LIN {X 0,Y 467.101,Z 440.554,A -85,B 0,C 180,E1 -7437.809,E2 -7437.809} C_VEL
LIN {X 0,Y 466.895,Z 445.866,A -85,B 0,C 180,E1 -7439.217,E2 -7439.217} C_VEL
LIN {X 0,Y 466.777,Z 448.845,A -85,B 0,C 180,E1 -7440.207,E2 -7440.207} C_VEL
LIN {X 0,Y 466.674,Z 451.155,A -85,B 0,C 180,E1 -7441.19,E2 -7441.19} C_VEL
LIN {X 0,Y 466.545,Z 453.69,A -85,B 0,C 180,E1 -7442.72,E2 -7442.72} C_VEL
LIN {X 0,Y 466.485,Z 454.874,A -85,B 0,C 180,E1 -7444.093,E2 -7444.093} C_VEL
LIN {X 0,Y 466.485,Z 455.129,A -85,B 0,C 180,E1 -7445.049,E2 -7445.049} C_VEL
LIN {X 0,Y 466.511,Z 454.294,A -85,B 0,C 180,E1 -7446.776,E2 -7446.776} C_VEL
LIN {X 0,Y 466.551,Z 452.966,A -85,B 0,C 180,E1 -7447.877,E2 -7447.877} C_VEL
LIN {X 0,Y 466.7,Z 450.858,A -85,B 0,C 180,E1 -7449.013,E2 -7449.013} C_VEL
LIN {X 0,Y 466.824,Z 447.854,A -85,B 0,C 180,E1 -7450.2,E2 -7450.2} C_VEL
LIN {X 0,Y 466.968,Z 443.277,A -85,B 0,C 180,E1 -7451.575,E2 -7451.575} C_VEL
LIN {X 0,Y 467.167,Z 437.426,A -85,B 0,C 180,E1 -7452.941,E2 -7452.941} C_VEL
LIN {X 0,Y 467.539,Z 430.017,A -85,B 0,C 180,E1 -7454.302,E2 -7454.302} C_VEL
LIN {X 0,Y 467.973,Z 420.781,A -85,B 0,C 180,E1 -7455.653,E2 -7455.653} C_VEL
LIN {X 0,Y 468.422,Z 411.25,A -85,B 0,C 180,E1 -7456.773,E2 -7456.773} C_VEL
LIN {X 0,Y 468.937,Z 400.379,A -85,B 0,C 180,E1 -7457.795,E2 -7457.795} C_VEL
LIN {X 0,Y 469.51,Z 388.647,A -85,B 0,C 180,E1 -7458.67,E2 -7458.67} C_VEL
LIN {X 0,Y 469.897,Z 377.126,A -85,B 0,C 180,E1 -7459.334,E2 -7459.334} C_VEL
LIN {X 0,Y 470.249,Z 364.286,A -85,B 0,C 180,E1 -7459.879,E2 -7459.879} C_VEL
LIN {X 0,Y 470.485,Z 351.401,A -85,B 0,C 180,E1 -7460.247,E2 -7460.247} C_VEL
LIN {X 0,Y 471.239,Z 259.051,A -85,B 0,C 180,E1 -7461.693,E2 -7461.693} C_VEL
LIN {X 0,Y 468.413,Z 244.23,A -85,B 0,C 180,E1 -7462.049,E2 -7462.049} C_VEL
LIN {X 0,Y 468.927,Z 230.528,A -85,B 0,C 180,E1 -7464.841,E2 -7464.841} C_VEL
LIN {X 0,Y 468.176,Z 224.517,A -85,B 0,C 180,E1 -7466.127,E2 -7466.127} C_VEL
LIN {X 0,Y 467.658,Z 221.234,A -85,B 0,C 180,E1 -7466.877,E2 -7466.877} C_VEL
LIN {X 0,Y 467.749,Z 221.221,A -85,B 0,C 180,E1 -7468.278,E2 -7468.278} C_VEL
LIN {X 0,Y 467.852,Z 221.207,A -85,B 0,C 180,E1 -7470,E2 -7470} C_VEL
LIN {X 0,Y 467.818,Z 221.207,A -85,B 0,C 180,E1 -7472.583,E2 -7472.583} C_VEL
LIN {X 0,Y 467.708,Z 221.224,A -85,B 0,C 180,E1 -7476.038,E2 -7476.038} C_VEL
LIN {X 0,Y 467.67,Z 221.226,A -85,B 0,C 180,E1 -7478.643,E2 -7478.643} C_VEL
LIN {X 0,Y 467.659,Z 221.229,A -85,B 0,C 180,E1 -7482.145,E2 -7482.145} C_VEL
LIN {X 0,Y 467.64,Z 221.237,A -85,B 0,C 180,E1 -7485.695,E2 -7485.695} C_VEL
LIN {X 0,Y 467.622,Z 221.236,A -85,B 0,C 180,E1 -7489.308,E2 -7489.308} C_VEL
LIN {X 0,Y 467.536,Z 221.245,A -85,B 0,C 180,E1 -7492.073,E2 -7492.073} C_VEL
LIN {X 0,Y 467.57,Z 221.241,A -85,B 0,C 180,E1 -7494.889,E2 -7494.889} C_VEL
LIN {X 0,Y 467.581,Z 221.243,A -85,B 0,C 180,E1 -7497.771,E2 -7497.771} C_VEL
LIN {X 0,Y 467.569,Z 221.242,A -85,B 0,C 180,E1 -7501.044,E2 -7501.044} C_VEL
LIN {X 0,Y 467.588,Z 221.238,A -85,B 0,C 180,E1 -7504.242,E2 -7504.242} C_VEL
LIN {X 0,Y 467.543,Z 221.245,A -85,B 0,C 180,E1 -7507.185,E2 -7507.185} C_VEL
LIN {X 0,Y 467.572,Z 221.24,A -85,B 0,C 180,E1 -7510.265,E2 -7510.265} C_VEL
LIN {X 0,Y 467.548,Z 221.246,A -85,B 0,C 180,E1 -7513.745,E2 -7513.745} C_VEL
LIN {X 0,Y 467.55,Z 221.243,A -85,B 0,C 180,E1 -7516.255,E2 -7516.255} C_VEL
LIN {X 0,Y 467.577,Z 221.241,A -85,B 0,C 180,E1 -7518.723,E2 -7518.723} C_VEL
LIN {X 0,Y 467.564,Z 221.242,A -85,B 0,C 180,E1 -7521.955,E2 -7521.955} C_VEL
LIN {X 0,Y 467.566,Z 221.243,A -85,B 0,C 180,E1 -7525.167,E2 -7525.167} C_VEL
LIN {X 0,Y 467.581,Z 221.24,A -85,B 0,C 180,E1 -7528.26,E2 -7528.26} C_VEL
LIN {X 0,Y 467.575,Z 221.242,A -85,B 0,C 180,E1 -7531.25,E2 -7531.25} C_VEL
LIN {X 0,Y 467.608,Z 221.236,A -85,B 0,C 180,E1 -7534.16,E2 -7534.16} C_VEL
LIN {X 0,Y 467.575,Z 221.242,A -85,B 0,C 180,E1 -7536.996,E2 -7536.996} C_VEL
LIN {X 0,Y 467.62,Z 221.236,A -85,B 0,C 180,E1 -7539.777,E2 -7539.777} C_VEL
LIN {X 0,Y 467.604,Z 221.238,A -85,B 0,C 180,E1 -7542.506,E2 -7542.506} C_VEL
LIN {X 0,Y 467.604,Z 221.239,A -85,B 0,C 180,E1 -7545.196,E2 -7545.196} C_VEL
LIN {X 0,Y 467.653,Z 221.231,A -85,B 0,C 180,E1 -7547.854,E2 -7547.854} C_VEL
LIN {X 0,Y 467.679,Z 221.23,A -85,B 0,C 180,E1 -7551.357,E2 -7551.357} C_VEL
LIN {X 0,Y 467.743,Z 221.22,A -85,B 0,C 180,E1 -7553.963,E2 -7553.963} C_VEL
LIN {X 0,Y 467.857,Z 221.207,A -85,B 0,C 180,E1 -7557.417,E2 -7557.417} C_VEL
LIN {X 0,Y 467.879,Z 221.202,A -85,B 0,C 180,E1 -7560,E2 -7560} C_VEL
LIN {X 0,Y 467.857,Z 221.208,A -85,B 0,C 180,E1 -7562.583,E2 -7562.583} C_VEL
LIN {X 0,Y 467.743,Z 221.219,A -85,B 0,C 180,E1 -7566.037,E2 -7566.037} C_VEL
LIN {X 0,Y 467.678,Z 221.232,A -85,B 0,C 180,E1 -7568.643,E2 -7568.643} C_VEL
LIN {X 0,Y 467.653,Z 221.231,A -85,B 0,C 180,E1 -7572.146,E2 -7572.146} C_VEL
LIN {X 0,Y 467.636,Z 221.233,A -85,B 0,C 180,E1 -7575.695,E2 -7575.695} C_VEL
LIN {X 0,Y 467.615,Z 221.239,A -85,B 0,C 180,E1 -7578.765,E2 -7578.765} C_VEL
LIN {X 0,Y 467.578,Z 221.241,A -85,B 0,C 180,E1 -7581.269,E2 -7581.269} C_VEL
LIN {X 0,Y 467.571,Z 221.24,A -85,B 0,C 180,E1 -7583.943,E2 -7583.943} C_VEL
LIN {X 0,Y 467.614,Z 221.238,A -85,B 0,C 180,E1 -7586.8,E2 -7586.8} C_VEL
LIN {X 0,Y 467.552,Z 221.242,A -85,B 0,C 180,E1 -7589.738,E2 -7589.738} C_VEL
LIN {X 0,Y 467.581,Z 221.243,A -85,B 0,C 180,E1 -7592.759,E2 -7592.759} C_VEL
LIN {X 0,Y 467.554,Z 221.242,A -85,B 0,C 180,E1 -7595.89,E2 -7595.89} C_VEL
LIN {X 0,Y 467.58,Z 221.24,A -85,B 0,C 180,E1 -7599.145,E2 -7599.145} C_VEL
LIN {X 0,Y 467.585,Z 221.244,A -85,B 0,C 180,E1 -7602.567,E2 -7602.567} C_VEL
LIN {X 0,Y 467.569,Z 221.241,A -85,B 0,C 180,E1 -7605.053,E2 -7605.053} C_VEL
LIN {X 0,Y 467.588,Z 221.237,A -85,B 0,C 180,E1 -7607.44,E2 -7607.44} C_VEL
LIN {X 0,Y 467.581,Z 221.241,A -85,B 0,C 180,E1 -7610.856,E2 -7610.856} C_VEL
LIN {X 0,Y 467.557,Z 221.244,A -85,B 0,C 180,E1 -7614.262,E2 -7614.262} C_VEL
LIN {X 0,Y 467.582,Z 221.238,A -85,B 0,C 180,E1 -7617.321,E2 -7617.321} C_VEL
LIN {X 0,Y 467.569,Z 221.246,A -85,B 0,C 180,E1 -7620.668,E2 -7620.668} C_VEL
LIN {X 0,Y 467.587,Z 221.244,A -85,B 0,C 180,E1 -7623.198,E2 -7623.198} C_VEL
LIN {X 0,Y 467.648,Z 221.415,A -85,B 0,C 180,E1 -7624.383,E2 -7624.383} C_VEL
LIN {X 0,Y 469.778,Z 233.014,A -85,B 0,C 180,E1 -7626.644,E2 -7626.644} C_VEL
LIN {X 0,Y 469.201,Z 246.955,A -85,B 0,C 180,E1 -7629.161,E2 -7629.161} C_VEL
LIN {X 0,Y 468.484,Z 264.68,A -85,B 0,C 180,E1 -7632.315,E2 -7632.315} C_VEL
LIN {X 0,Y 468.326,Z 268.709,A -85,B 0,C 180,E1 -7633.001,E2 -7633.001} C_VEL
LIN {X 0,Y 471.206,Z 287.43,A -85,B 0,C 180,E1 -7633.4,E2 -7633.4} C_VEL
LIN {X 0,Y 470.468,Z 376.468,A -85,B 0,C 180,E1 -7634.79,E2 -7634.79} C_VEL
LIN {X 0,Y 470.15,Z 389.788,A -85,B 0,C 180,E1 -7635.168,E2 -7635.168} C_VEL
LIN {X 0,Y 469.684,Z 402.549,A -85,B 0,C 180,E1 -7635.706,E2 -7635.706} C_VEL
LIN {X 0,Y 469.237,Z 413.892,A -85,B 0,C 180,E1 -7636.356,E2 -7636.356} C_VEL
LIN {X 0,Y 468.679,Z 425.815,A -85,B 0,C 180,E1 -7637.241,E2 -7637.241} C_VEL
LIN {X 0,Y 468.248,Z 436.107,A -85,B 0,C 180,E1 -7638.2,E2 -7638.2} C_VEL
LIN {X 0,Y 467.781,Z 444.702,A -85,B 0,C 180,E1 -7639.176,E2 -7639.176} C_VEL
LIN {X 0,Y 467.436,Z 452.63,A -85,B 0,C 180,E1 -7640.262,E2 -7640.262} C_VEL
LIN {X 0,Y 467.111,Z 460.375,A -85,B 0,C 180,E1 -7641.565,E2 -7641.565} C_VEL
LIN {X 0,Y 466.852,Z 467.499,A -85,B 0,C 180,E1 -7643.083,E2 -7643.083} C_VEL
LIN {X 0,Y 466.76,Z 472.241,A -85,B 0,C 180,E1 -7644.384,E2 -7644.384} C_VEL
LIN {X 0,Y 466.646,Z 475.861,A -85,B 0,C 180,E1 -7645.682,E2 -7645.682} C_VEL
LIN {X 0,Y 466.688,Z 477.732,A -85,B 0,C 180,E1 -7646.547,E2 -7646.547} C_VEL
LIN {X 0,Y 466.662,Z 479.133,A -85,B 0,C 180,E1 -7647.411,E2 -7647.411} C_VEL
LIN {X 0,Y 466.619,Z 480.737,A -85,B 0,C 180,E1 -7649.137,E2 -7649.137} C_VEL
LIN {X 0,Y 466.6,Z 480.953,A -85,B 0,C 180,E1 -7650,E2 -7650} C_VEL
LIN {X 0,Y 466.619,Z 480.735,A -85,B 0,C 180,E1 -7650.863,E2 -7650.863} C_VEL
LIN {X 0,Y 466.662,Z 479.123,A -85,B 0,C 180,E1 -7652.59,E2 -7652.59} C_VEL
LIN {X 0,Y 466.688,Z 477.721,A -85,B 0,C 180,E1 -7653.454,E2 -7653.454} C_VEL
LIN {X 0,Y 466.688,Z 474.771,A -85,B 0,C 180,E1 -7654.751,E2 -7654.751} C_VEL
LIN {X 0,Y 466.75,Z 470.782,A -85,B 0,C 180,E1 -7656.05,E2 -7656.05} C_VEL
LIN {X 0,Y 466.942,Z 464.65,A -85,B 0,C 180,E1 -7657.568,E2 -7657.568} C_VEL
LIN {X 0,Y 467.217,Z 457.952,A -85,B 0,C 180,E1 -7658.87,E2 -7658.87} C_VEL
LIN {X 0,Y 467.546,Z 449.643,A -85,B 0,C 180,E1 -7660.173,E2 -7660.173} C_VEL
LIN {X 0,Y 468.016,Z 441.127,A -85,B 0,C 180,E1 -7661.257,E2 -7661.257} C_VEL
LIN {X 0,Y 468.511,Z 431.038,A -85,B 0,C 180,E1 -7662.302,E2 -7662.302} C_VEL
LIN {X 0,Y 468.935,Z 420.195,A -85,B 0,C 180,E1 -7663.212,E2 -7663.212} C_VEL
LIN {X 0,Y 469.459,Z 408.784,A -85,B 0,C 180,E1 -7663.969,E2 -7663.969} C_VEL
LIN {X 0,Y 469.892,Z 397.043,A -85,B 0,C 180,E1 -7664.564,E2 -7664.564} C_VEL
LIN {X 0,Y 470.35,Z 383.529,A -85,B 0,C 180,E1 -7665.047,E2 -7665.047} C_VEL
LIN {X 0,Y 470.646,Z 370.034,A -85,B 0,C 180,E1 -7665.343,E2 -7665.343} C_VEL
LIN {X 0,Y 471.145,Z 285.886,A -85,B 0,C 180,E1 -7666.649,E2 -7666.649} C_VEL
LIN {X 0,Y 468.3,Z 268.124,A -85,B 0,C 180,E1 -7667.05,E2 -7667.05} C_VEL
LIN {X 0,Y 468.908,Z 251.671,A -85,B 0,C 180,E1 -7669.936,E2 -7669.936} C_VEL
LIN {X 0,Y 469.636,Z 234.97,A -85,B 0,C 180,E1 -7672.898,E2 -7672.898} C_VEL
LIN {X 0,Y 469.472,Z 231.104,A -85,B 0,C 180,E1 -7673.606,E2 -7673.606} C_VEL
LIN {X 0,Y 467.615,Z 221.24,A -85,B 0,C 180,E1 -7675.512,E2 -7675.512} C_VEL
LIN {X 0,Y 467.617,Z 221.239,A -85,B 0,C 180,E1 -7677.769,E2 -7677.769} C_VEL
LIN {X 0,Y 467.569,Z 221.245,A -85,B 0,C 180,E1 -7681.045,E2 -7681.045} C_VEL
LIN {X 0,Y 467.589,Z 221.238,A -85,B 0,C 180,E1 -7684.242,E2 -7684.242} C_VEL
LIN {X 0,Y 467.543,Z 221.249,A -85,B 0,C 180,E1 -7687.185,E2 -7687.185} C_VEL
LIN {X 0,Y 467.575,Z 221.237,A -85,B 0,C 180,E1 -7690.265,E2 -7690.265} C_VEL
LIN {X 0,Y 467.587,Z 221.237,A -85,B 0,C 180,E1 -7692.567,E2 -7692.567} C_VEL
LIN {X 0,Y 467.571,Z 221.244,A -85,B 0,C 180,E1 -7695.053,E2 -7695.053} C_VEL
LIN {X 0,Y 467.589,Z 221.239,A -85,B 0,C 180,E1 -7697.44,E2 -7697.44} C_VEL
LIN {X 0,Y 467.576,Z 221.242,A -85,B 0,C 180,E1 -7700.855,E2 -7700.855} C_VEL
LIN {X 0,Y 467.562,Z 221.238,A -85,B 0,C 180,E1 -7704.26,E2 -7704.26} C_VEL
LIN {X 0,Y 467.581,Z 221.24,A -85,B 0,C 180,E1 -7707.321,E2 -7707.321} C_VEL
LIN {X 0,Y 467.57,Z 221.241,A -85,B 0,C 180,E1 -7710.667,E2 -7710.667} C_VEL
LIN {X 0,Y 467.616,Z 221.237,A -85,B 0,C 180,E1 -7713.2,E2 -7713.2} C_VEL
LIN {X 0,Y 467.592,Z 221.236,A -85,B 0,C 180,E1 -7716.468,E2 -7716.468} C_VEL
LIN {X 0,Y 467.622,Z 221.232,A -85,B 0,C 180,E1 -7719.777,E2 -7719.777} C_VEL
LIN {X 0,Y 467.606,Z 221.233,A -85,B 0,C 180,E1 -7722.507,E2 -7722.507} C_VEL
LIN {X 0,Y 467.606,Z 221.234,A -85,B 0,C 180,E1 -7725.196,E2 -7725.196} C_VEL
LIN {X 0,Y 467.655,Z 221.227,A -85,B 0,C 180,E1 -7727.855,E2 -7727.855} C_VEL
LIN {X 0,Y 467.681,Z 221.226,A -85,B 0,C 180,E1 -7731.357,E2 -7731.357} C_VEL
LIN {X 0,Y 467.734,Z 221.217,A -85,B 0,C 180,E1 -7733.963,E2 -7733.963} C_VEL
LIN {X 0,Y 467.859,Z 221.204,A -85,B 0,C 180,E1 -7737.417,E2 -7737.417} C_VEL
LIN {X 0,Y 467.881,Z 221.196,A -85,B 0,C 180,E1 -7740,E2 -7740} C_VEL
LIN {X 0,Y 467.858,Z 221.208,A -85,B 0,C 180,E1 -7742.583,E2 -7742.583} C_VEL
LIN {X 0,Y 467.734,Z 221.219,A -85,B 0,C 180,E1 -7746.038,E2 -7746.038} C_VEL
LIN {X 0,Y 467.681,Z 221.228,A -85,B 0,C 180,E1 -7748.643,E2 -7748.643} C_VEL
LIN {X 0,Y 467.655,Z 221.226,A -85,B 0,C 180,E1 -7752.146,E2 -7752.146} C_VEL
LIN {X 0,Y 467.639,Z 221.228,A -85,B 0,C 180,E1 -7755.695,E2 -7755.695} C_VEL
LIN {X 0,Y 467.617,Z 221.238,A -85,B 0,C 180,E1 -7758.765,E2 -7758.765} C_VEL
LIN {X 0,Y 467.58,Z 221.238,A -85,B 0,C 180,E1 -7761.268,E2 -7761.268} C_VEL
LIN {X 0,Y 467.563,Z 221.24,A -85,B 0,C 180,E1 -7763.944,E2 -7763.944} C_VEL
LIN {X 0,Y 467.565,Z 221.245,A -85,B 0,C 180,E1 -7766.804,E2 -7766.804} C_VEL
LIN {X 0,Y 467.547,Z 221.24,A -85,B 0,C 180,E1 -7769.739,E2 -7769.739} C_VEL
LIN {X 0,Y 467.579,Z 221.243,A -85,B 0,C 180,E1 -7772.759,E2 -7772.759} C_VEL
LIN {X 0,Y 467.549,Z 221.246,A -85,B 0,C 180,E1 -7775.89,E2 -7775.89} C_VEL
LIN {X 0,Y 467.547,Z 221.245,A -85,B 0,C 180,E1 -7779.149,E2 -7779.149} C_VEL
LIN {X 0,Y 467.564,Z 221.243,A -85,B 0,C 180,E1 -7781.405,E2 -7781.405} C_VEL
LIN {X 0,Y 467.564,Z 221.31,A -85,B 0,C 180,E1 -7783.521,E2 -7783.521} C_VEL
LIN {X 0,Y 468.843,Z 228.525,A -85,B 0,C 180,E1 -7785.001,E2 -7785.001} C_VEL
LIN {X 0,Y 468.462,Z 244.324,A -85,B 0,C 180,E1 -7788.025,E2 -7788.025} C_VEL
LIN {X 0,Y 471.369,Z 259.441,A -85,B 0,C 180,E1 -7788.378,E2 -7788.378} C_VEL
LIN {X 0,Y 470.565,Z 351.674,A -85,B 0,C 180,E1 -7789.824,E2 -7789.824} C_VEL
LIN {X 0,Y 470.284,Z 365.391,A -85,B 0,C 180,E1 -7790.223,E2 -7790.223} C_VEL
LIN {X 0,Y 469.973,Z 377.504,A -85,B 0,C 180,E1 -7790.747,E2 -7790.747} C_VEL
LIN {X 0,Y 469.481,Z 389.628,A -85,B 0,C 180,E1 -7791.456,E2 -7791.456} C_VEL
LIN {X 0,Y 469.023,Z 400.201,A -85,B 0,C 180,E1 -7792.251,E2 -7792.251} C_VEL
LIN {X 0,Y 468.509,Z 411.002,A -85,B 0,C 180,E1 -7793.262,E2 -7793.262} C_VEL
LIN {X 0,Y 468.031,Z 420.88,A -85,B 0,C 180,E1 -7794.42,E2 -7794.42} C_VEL
LIN {X 0,Y 467.78,Z 426.185,A -85,B 0,C 180,E1 -7795.161,E2 -7795.161} C_VEL
LIN {X 0,Y 467.008,Z 429.892,A -85,B 0,C 180,E1 -7795.717,E2 -7795.717} C_VEL
LIN {X 0,Y 463.897,Z 435.547,A -85,B 0,C 180,E1 -7796.645,E2 -7796.645} C_VEL
LIN {X 0,Y 460.752,Z 440.515,A -85,B 0,C 180,E1 -7797.639,E2 -7797.639} C_VEL
LIN {X 0,Y 459.944,Z 443.146,A -85,B 0,C 180,E1 -7798.292,E2 -7798.292} C_VEL
LIN {X 0,Y 459.792,Z 447.857,A -85,B 0,C 180,E1 -7799.708,E2 -7799.708} C_VEL
LIN {X 0,Y 459.658,Z 450.452,A -85,B 0,C 180,E1 -7800.708,E2 -7800.708} C_VEL
LIN {X 0,Y 459.525,Z 452.445,A -85,B 0,C 180,E1 -7801.698,E2 -7801.698} C_VEL
LIN {X 0,Y 459.464,Z 453.893,A -85,B 0,C 180,E1 -7802.685,E2 -7802.685} C_VEL
LIN {X 0,Y 459.408,Z 454.848,A -85,B 0,C 180,E1 -7803.664,E2 -7803.664} C_VEL
LIN {X 0,Y 459.416,Z 455.261,A -85,B 0,C 180,E1 -7804.638,E2 -7804.638} C_VEL
LIN {X 0,Y 459.386,Z 455.226,A -85,B 0,C 180,E1 -7805.603,E2 -7805.603} C_VEL
LIN {X 0,Y 459.418,Z 454.657,A -85,B 0,C 180,E1 -7806.615,E2 -7806.615} C_VEL
LIN {X 0,Y 459.429,Z 453.7,A -85,B 0,C 180,E1 -7807.516,E2 -7807.516} C_VEL
LIN {X 0,Y 459.585,Z 451.44,A -85,B 0,C 180,E1 -7808.879,E2 -7808.879} C_VEL
LIN {X 0,Y 459.752,Z 447.841,A -85,B 0,C 180,E1 -7810.348,E2 -7810.348} C_VEL
LIN {X 0,Y 459.909,Z 443.083,A -85,B 0,C 180,E1 -7811.777,E2 -7811.777} C_VEL
LIN {X 0,Y 460.145,Z 437.274,A -85,B 0,C 180,E1 -7813.13,E2 -7813.13} C_VEL
LIN {X 0,Y 460.539,Z 429.763,A -85,B 0,C 180,E1 -7814.511,E2 -7814.511} C_VEL
LIN {X 0,Y 461.007,Z 420.437,A -85,B 0,C 180,E1 -7815.882,E2 -7815.882} C_VEL
LIN {X 0,Y 461.567,Z 410.599,A -85,B 0,C 180,E1 -7817.032,E2 -7817.032} C_VEL
LIN {X 0,Y 462.057,Z 399.903,A -85,B 0,C 180,E1 -7818.039,E2 -7818.039} C_VEL
LIN {X 0,Y 462.564,Z 389.426,A -85,B 0,C 180,E1 -7818.83,E2 -7818.83} C_VEL
LIN {X 0,Y 463.044,Z 376.849,A -85,B 0,C 180,E1 -7819.567,E2 -7819.567} C_VEL
LIN {X 0,Y 463.389,Z 363.758,A -85,B 0,C 180,E1 -7820.124,E2 -7820.124} C_VEL
LIN {X 0,Y 463.647,Z 351.397,A -85,B 0,C 180,E1 -7820.475,E2 -7820.475} C_VEL
LIN {X 0,Y 464.461,Z 260.073,A -85,B 0,C 180,E1 -7821.924,E2 -7821.924} C_VEL
LIN {X 0,Y 461.465,Z 244.435,A -85,B 0,C 180,E1 -7822.302,E2 -7822.302} C_VEL
LIN {X 0,Y 461.918,Z 230.419,A -85,B 0,C 180,E1 -7825.2,E2 -7825.2} C_VEL
LIN {X 0,Y 460.644,Z 222.108,A -85,B 0,C 180,E1 -7827.048,E2 -7827.048} C_VEL
LIN {X 0,Y 460.822,Z 222.083,A -85,B 0,C 180,E1 -7830,E2 -7830} C_VEL
LIN {X 0,Y 460.762,Z 222.086,A -85,B 0,C 180,E1 -7832.623,E2 -7832.623} C_VEL
LIN {X 0,Y 460.674,Z 222.1,A -85,B 0,C 180,E1 -7836.13,E2 -7836.13} C_VEL
LIN {X 0,Y 460.62,Z 222.105,A -85,B 0,C 180,E1 -7838.776,E2 -7838.776} C_VEL
LIN {X 0,Y 460.6,Z 222.108,A -85,B 0,C 180,E1 -7842.435,E2 -7842.435} C_VEL
LIN {X 0,Y 460.581,Z 222.113,A -85,B 0,C 180,E1 -7845.988,E2 -7845.988} C_VEL
LIN {X 0,Y 460.569,Z 222.118,A -85,B 0,C 180,E1 -7849.615,E2 -7849.615} C_VEL
LIN {X 0,Y 460.512,Z 222.119,A -85,B 0,C 180,E1 -7852.428,E2 -7852.428} C_VEL
LIN {X 0,Y 460.549,Z 222.119,A -85,B 0,C 180,E1 -7855.796,E2 -7855.796} C_VEL
LIN {X 0,Y 460.528,Z 222.118,A -85,B 0,C 180,E1 -7858.234,E2 -7858.234} C_VEL
LIN {X 0,Y 460.521,Z 222.12,A -85,B 0,C 180,E1 -7861.282,E2 -7861.282} C_VEL
LIN {X 0,Y 460.531,Z 222.117,A -85,B 0,C 180,E1 -7864.505,E2 -7864.505} C_VEL
LIN {X 0,Y 460.499,Z 222.126,A -85,B 0,C 180,E1 -7867.623,E2 -7867.623} C_VEL
LIN {X 0,Y 460.536,Z 222.117,A -85,B 0,C 180,E1 -7870.268,E2 -7870.268} C_VEL
LIN {X 0,Y 460.508,Z 222.123,A -85,B 0,C 180,E1 -7873.374,E2 -7873.374} C_VEL
LIN {X 0,Y 460.496,Z 222.123,A -85,B 0,C 180,E1 -7876.624,E2 -7876.624} C_VEL
LIN {X 0,Y 460.538,Z 222.12,A -85,B 0,C 180,E1 -7879.731,E2 -7879.731} C_VEL
LIN {X 0,Y 460.499,Z 222.122,A -85,B 0,C 180,E1 -7882.523,E2 -7882.523} C_VEL
LIN {X 0,Y 460.547,Z 222.119,A -85,B 0,C 180,E1 -7885.624,E2 -7885.624} C_VEL
LIN {X 0,Y 460.535,Z 222.119,A -85,B 0,C 180,E1 -7888.744,E2 -7888.744} C_VEL
LIN {X 0,Y 460.579,Z 222.112,A -85,B 0,C 180,E1 -7892.253,E2 -7892.253} C_VEL
LIN {X 0,Y 460.557,Z 222.117,A -85,B 0,C 180,E1 -7894.705,E2 -7894.705} C_VEL
LIN {X 0,Y 460.509,Z 222.124,A -85,B 0,C 180,E1 -7897.571,E2 -7897.571} C_VEL
LIN {X 0,Y 460.566,Z 222.114,A -85,B 0,C 180,E1 -7900.384,E2 -7900.384} C_VEL
LIN {X 0,Y 460.562,Z 222.115,A -85,B 0,C 180,E1 -7903.146,E2 -7903.146} C_VEL
LIN {X 0,Y 460.552,Z 222.116,A -85,B 0,C 180,E1 -7905.868,E2 -7905.868} C_VEL
LIN {X 0,Y 460.609,Z 222.11,A -85,B 0,C 180,E1 -7908.559,E2 -7908.559} C_VEL
LIN {X 0,Y 460.692,Z 222.098,A -85,B 0,C 180,E1 -7912.108,E2 -7912.108} C_VEL
LIN {X 0,Y 460.696,Z 222.1,A -85,B 0,C 180,E1 -7914.748,E2 -7914.748} C_VEL
LIN {X 0,Y 460.822,Z 222.083,A -85,B 0,C 180,E1 -7917.378,E2 -7917.378} C_VEL
LIN {X 0,Y 460.85,Z 222.078,A -85,B 0,C 180,E1 -7920,E2 -7920} C_VEL
LIN {X 0,Y 460.822,Z 222.085,A -85,B 0,C 180,E1 -7922.622,E2 -7922.622} C_VEL
LIN {X 0,Y 460.709,Z 222.096,A -85,B 0,C 180,E1 -7926.13,E2 -7926.13} C_VEL
LIN {X 0,Y 460.625,Z 222.109,A -85,B 0,C 180,E1 -7928.776,E2 -7928.776} C_VEL
LIN {X 0,Y 460.61,Z 222.11,A -85,B 0,C 180,E1 -7932.445,E2 -7932.445} C_VEL
LIN {X 0,Y 460.597,Z 222.109,A -85,B 0,C 180,E1 -7935.998,E2 -7935.998} C_VEL
LIN {X 0,Y 460.568,Z 222.115,A -85,B 0,C 180,E1 -7938.902,E2 -7938.902} C_VEL
LIN {X 0,Y 460.513,Z 222.121,A -85,B 0,C 180,E1 -7941.486,E2 -7941.486} C_VEL
LIN {X 0,Y 460.54,Z 222.118,A -85,B 0,C 180,E1 -7944.332,E2 -7944.332} C_VEL
LIN {X 0,Y 460.57,Z 222.113,A -85,B 0,C 180,E1 -7947.244,E2 -7947.244} C_VEL
LIN {X 0,Y 460.508,Z 222.122,A -85,B 0,C 180,E1 -7950.24,E2 -7950.24} C_VEL
LIN {X 0,Y 460.527,Z 222.118,A -85,B 0,C 180,E1 -7953.325,E2 -7953.325} C_VEL
LIN {X 0,Y 460.476,Z 222.129,A -85,B 0,C 180,E1 -7956.53,E2 -7956.53} C_VEL
LIN {X 0,Y 460.53,Z 222.117,A -85,B 0,C 180,E1 -7959.863,E2 -7959.863} C_VEL
LIN {X 0,Y 460.512,Z 222.121,A -85,B 0,C 180,E1 -7962.901,E2 -7962.901} C_VEL
LIN {X 0,Y 460.51,Z 222.119,A -85,B 0,C 180,E1 -7965.831,E2 -7965.831} C_VEL
LIN {X 0,Y 460.53,Z 222.118,A -85,B 0,C 180,E1 -7968.989,E2 -7968.989} C_VEL
LIN {X 0,Y 460.524,Z 222.117,A -85,B 0,C 180,E1 -7971.267,E2 -7971.267} C_VEL
LIN {X 0,Y 460.508,Z 222.126,A -85,B 0,C 180,E1 -7974.555,E2 -7974.555} C_VEL
LIN {X 0,Y 460.531,Z 222.115,A -85,B 0,C 180,E1 -7977.716,E2 -7977.716} C_VEL
LIN {X 0,Y 460.539,Z 222.121,A -85,B 0,C 180,E1 -7980.769,E2 -7980.769} C_VEL
LIN {X 0,Y 460.546,Z 222.121,A -85,B 0,C 180,E1 -7983.734,E2 -7983.734} C_VEL
LIN {X 0,Y 460.575,Z 222.201,A -85,B 0,C 180,E1 -7984.153,E2 -7984.153} C_VEL
LIN {X 0,Y 462.801,Z 234.066,A -85,B 0,C 180,E1 -7986.508,E2 -7986.508} C_VEL
LIN {X 0,Y 462.24,Z 248.01,A -85,B 0,C 180,E1 -7989.066,E2 -7989.066} C_VEL
LIN {X 0,Y 461.464,Z 265.729,A -85,B 0,C 180,E1 -7992.266,E2 -7992.266} C_VEL
LIN {X 0,Y 461.339,Z 268.541,A -85,B 0,C 180,E1 -7992.741,E2 -7992.741} C_VEL
LIN {X 0,Y 464.399,Z 287.867,A -85,B 0,C 180,E1 -7993.165,E2 -7993.165} C_VEL
LIN {X 0,Y 463.577,Z 377.159,A -85,B 0,C 180,E1 -7994.587,E2 -7994.587} C_VEL
LIN {X 0,Y 463.193,Z 390.942,A -85,B 0,C 180,E1 -7994.996,E2 -7994.996} C_VEL
LIN {X 0,Y 462.761,Z 403.327,A -85,B 0,C 180,E1 -7995.544,E2 -7995.544} C_VEL
LIN {X 0,Y 462.244,Z 415.198,A -85,B 0,C 180,E1 -7996.257,E2 -7996.257} C_VEL
LIN {X 0,Y 461.692,Z 426.438,A -85,B 0,C 180,E1 -7997.122,E2 -7997.122} C_VEL
LIN {X 0,Y 461.218,Z 436.918,A -85,B 0,C 180,E1 -7998.129,E2 -7998.129} C_VEL
LIN {X 0,Y 460.682,Z 446.162,A -85,B 0,C 180,E1 -7999.229,E2 -7999.229} C_VEL
LIN {X 0,Y 460.265,Z 455.154,A -85,B 0,C 180,E1 -8000.553,E2 -8000.553} C_VEL
LIN {X 0,Y 459.951,Z 462.395,A -85,B 0,C 180,E1 -8001.875,E2 -8001.875} C_VEL
LIN {X 0,Y 459.743,Z 468.46,A -85,B 0,C 180,E1 -8003.273,E2 -8003.273} C_VEL
LIN {X 0,Y 459.649,Z 473.351,A -85,B 0,C 180,E1 -8004.736,E2 -8004.736} C_VEL
LIN {X 0,Y 459.563,Z 475.655,A -85,B 0,C 180,E1 -8005.615,E2 -8005.615} C_VEL
LIN {X 0,Y 459.583,Z 477.528,A -85,B 0,C 180,E1 -8006.493,E2 -8006.493} C_VEL
LIN {X 0,Y 459.584,Z 478.932,A -85,B 0,C 180,E1 -8007.371,E2 -8007.371} C_VEL
LIN {X 0,Y 459.522,Z 480.539,A -85,B 0,C 180,E1 -8009.124,E2 -8009.124} C_VEL
LIN {X 0,Y 459.531,Z 480.757,A -85,B 0,C 180,E1 -8010,E2 -8010} C_VEL
LIN {X 0,Y 459.522,Z 480.54,A -85,B 0,C 180,E1 -8010.876,E2 -8010.876} C_VEL
LIN {X 0,Y 459.584,Z 478.93,A -85,B 0,C 180,E1 -8012.63,E2 -8012.63} C_VEL
LIN {X 0,Y 459.583,Z 477.528,A -85,B 0,C 180,E1 -8013.507,E2 -8013.507} C_VEL
LIN {X 0,Y 459.616,Z 474.581,A -85,B 0,C 180,E1 -8014.824,E2 -8014.824} C_VEL
LIN {X 0,Y 459.714,Z 469.56,A -85,B 0,C 180,E1 -8016.431,E2 -8016.431} C_VEL
LIN {X 0,Y 459.901,Z 463.447,A -85,B 0,C 180,E1 -8017.905,E2 -8017.905} C_VEL
LIN {X 0,Y 460.212,Z 456.525,A -85,B 0,C 180,E1 -8019.227,E2 -8019.227} C_VEL
LIN {X 0,Y 460.503,Z 449.458,A -85,B 0,C 180,E1 -8020.33,E2 -8020.33} C_VEL
LIN {X 0,Y 461.029,Z 440.946,A -85,B 0,C 180,E1 -8021.43,E2 -8021.43} C_VEL
LIN {X 0,Y 461.557,Z 431.024,A -85,B 0,C 180,E1 -8022.475,E2 -8022.475} C_VEL
LIN {X 0,Y 462.011,Z 420.022,A -85,B 0,C 180,E1 -8023.414,E2 -8023.414} C_VEL
LIN {X 0,Y 462.55,Z 408.618,A -85,B 0,C 180,E1 -8024.182,E2 -8024.182} C_VEL
LIN {X 0,Y 463.021,Z 396.894,A -85,B 0,C 180,E1 -8024.785,E2 -8024.785} C_VEL
LIN {X 0,Y 463.504,Z 383.404,A -85,B 0,C 180,E1 -8025.275,E2 -8025.275} C_VEL
LIN {X 0,Y 463.818,Z 369.991,A -85,B 0,C 180,E1 -8025.574,E2 -8025.574} C_VEL
LIN {X 0,Y 464.358,Z 286.812,A -85,B 0,C 180,E1 -8026.886,E2 -8026.886} C_VEL
LIN {X 0,Y 461.349,Z 267.883,A -85,B 0,C 180,E1 -8027.327,E2 -8027.327} C_VEL
LIN {X 0,Y 462.003,Z 251.476,A -85,B 0,C 180,E1 -8030.247,E2 -8030.247} C_VEL
LIN {X 0,Y 462.779,Z 234.798,A -85,B 0,C 180,E1 -8033.257,E2 -8033.257} C_VEL
LIN {X 0,Y 461.519,Z 227.044,A -85,B 0,C 180,E1 -8034.757,E2 -8034.757} C_VEL
LIN {X 0,Y 460.559,Z 222.118,A -85,B 0,C 180,E1 -8035.743,E2 -8035.743} C_VEL
LIN {X 0,Y 460.55,Z 222.117,A -85,B 0,C 180,E1 -8038.233,E2 -8038.233} C_VEL
LIN {X 0,Y 460.522,Z 222.125,A -85,B 0,C 180,E1 -8041.283,E2 -8041.283} C_VEL
LIN {X 0,Y 460.532,Z 222.118,A -85,B 0,C 180,E1 -8044.505,E2 -8044.505} C_VEL
LIN {X 0,Y 460.499,Z 222.123,A -85,B 0,C 180,E1 -8047.623,E2 -8047.623} C_VEL
LIN {X 0,Y 460.539,Z 222.114,A -85,B 0,C 180,E1 -8050.269,E2 -8050.269} C_VEL
LIN {X 0,Y 460.509,Z 222.126,A -85,B 0,C 180,E1 -8053.374,E2 -8053.374} C_VEL
LIN {X 0,Y 460.5,Z 222.122,A -85,B 0,C 180,E1 -8056.625,E2 -8056.625} C_VEL
LIN {X 0,Y 460.539,Z 222.117,A -85,B 0,C 180,E1 -8059.731,E2 -8059.731} C_VEL
LIN {X 0,Y 460.5,Z 222.119,A -85,B 0,C 180,E1 -8062.523,E2 -8062.523} C_VEL
LIN {X 0,Y 460.548,Z 222.115,A -85,B 0,C 180,E1 -8065.624,E2 -8065.624} C_VEL
LIN {X 0,Y 460.537,Z 222.115,A -85,B 0,C 180,E1 -8068.744,E2 -8068.744} C_VEL
LIN {X 0,Y 460.581,Z 222.107,A -85,B 0,C 180,E1 -8072.254,E2 -8072.254} C_VEL
LIN {X 0,Y 460.558,Z 222.115,A -85,B 0,C 180,E1 -8074.705,E2 -8074.705} C_VEL
LIN {X 0,Y 460.51,Z 222.119,A -85,B 0,C 180,E1 -8077.571,E2 -8077.571} C_VEL
LIN {X 0,Y 460.568,Z 222.111,A -85,B 0,C 180,E1 -8080.384,E2 -8080.384} C_VEL
LIN {X 0,Y 460.563,Z 222.117,A -85,B 0,C 180,E1 -8083.146,E2 -8083.146} C_VEL
LIN {X 0,Y 460.555,Z 222.107,A -85,B 0,C 180,E1 -8085.868,E2 -8085.868} C_VEL
LIN {X 0,Y 460.61,Z 222.108,A -85,B 0,C 180,E1 -8088.559,E2 -8088.559} C_VEL
LIN {X 0,Y 460.694,Z 222.094,A -85,B 0,C 180,E1 -8092.109,E2 -8092.109} C_VEL
LIN {X 0,Y 460.693,Z 222.098,A -85,B 0,C 180,E1 -8094.748,E2 -8094.748} C_VEL
LIN {X 0,Y 460.824,Z 222.081,A -85,B 0,C 180,E1 -8097.378,E2 -8097.378} C_VEL
LIN {X 0,Y 460.852,Z 222.071,A -85,B 0,C 180,E1 -8100,E2 -8100} C_VEL
LIN {X 0,Y 460.823,Z 222.085,A -85,B 0,C 180,E1 -8102.622,E2 -8102.622} C_VEL
LIN {X 0,Y 460.7,Z 222.095,A -85,B 0,C 180,E1 -8106.13,E2 -8106.13} C_VEL
LIN {X 0,Y 460.628,Z 222.107,A -85,B 0,C 180,E1 -8108.776,E2 -8108.776} C_VEL
LIN {X 0,Y 460.613,Z 222.106,A -85,B 0,C 180,E1 -8112.445,E2 -8112.445} C_VEL
LIN {X 0,Y 460.6,Z 222.106,A -85,B 0,C 180,E1 -8115.998,E2 -8115.998} C_VEL
LIN {X 0,Y 460.57,Z 222.116,A -85,B 0,C 180,E1 -8118.902,E2 -8118.902} C_VEL
LIN {X 0,Y 460.515,Z 222.117,A -85,B 0,C 180,E1 -8121.486,E2 -8121.486} C_VEL
LIN {X 0,Y 460.53,Z 222.119,A -85,B 0,C 180,E1 -8124.333,E2 -8124.333} C_VEL
LIN {X 0,Y 460.534,Z 222.117,A -85,B 0,C 180,E1 -8127.246,E2 -8127.246} C_VEL
LIN {X 0,Y 460.507,Z 222.121,A -85,B 0,C 180,E1 -8130.24,E2 -8130.24} C_VEL
LIN {X 0,Y 460.519,Z 222.12,A -85,B 0,C 180,E1 -8133.326,E2 -8133.326} C_VEL
LIN {X 0,Y 460.465,Z 222.132,A -85,B 0,C 180,E1 -8136.531,E2 -8136.531} C_VEL
LIN {X 0,Y 460.511,Z 222.122,A -85,B 0,C 180,E1 -8139.865,E2 -8139.865} C_VEL
LIN {X 0,Y 460.52,Z 222.123,A -85,B 0,C 180,E1 -8143.222,E2 -8143.222} C_VEL
LIN {X 0,Y 460.564,Z 222.384,A -85,B 0,C 180,E1 -8143.368,E2 -8143.368} C_VEL
LIN {X 0,Y 461.929,Z 230.208,A -85,B 0,C 180,E1 -8144.985,E2 -8144.985} C_VEL
LIN {X 0,Y 461.504,Z 244.26,A -85,B 0,C 180,E1 -8147.729,E2 -8147.729} C_VEL
LIN {X 0,Y 464.597,Z 260.384,A -85,B 0,C 180,E1 -8148.134,E2 -8148.134} C_VEL
LIN {X 0,Y 463.748,Z 351.503,A -85,B 0,C 180,E1 -8149.584,E2 -8149.584} C_VEL
LIN {X 0,Y 463.438,Z 365.072,A -85,B 0,C 180,E1 -8149.978,E2 -8149.978} C_VEL
LIN {X 0,Y 463.079,Z 377.362,A -85,B 0,C 180,E1 -8150.51,E2 -8150.51} C_VEL
LIN {X 0,Y 462.605,Z 389.448,A -85,B 0,C 180,E1 -8151.221,E2 -8151.221} C_VEL
LIN {X 0,Y 462.054,Z 401.471,A -85,B 0,C 180,E1 -8152.145,E2 -8152.145} C_VEL
LIN {X 0,Y 461.524,Z 411.961,A -85,B 0,C 180,E1 -8153.159,E2 -8153.159} C_VEL
LIN {X 0,Y 460.996,Z 421.793,A -85,B 0,C 180,E1 -8154.351,E2 -8154.351} C_VEL
LIN {X 0,Y 460.55,Z 430.286,A -85,B 0,C 180,E1 -8155.624,E2 -8155.624} C_VEL
LIN {X 0,Y 460.181,Z 437.34,A -85,B 0,C 180,E1 -8156.933,E2 -8156.933} C_VEL
LIN {X 0,Y 459.944,Z 443.146,A -85,B 0,C 180,E1 -8158.292,E2 -8158.292} C_VEL
LIN {X 0,Y 459.163,Z 445.588,A -85,B 0,C 180,E1 -8158.96,E2 -8158.96} C_VEL
LIN {X 0,Y 456.126,Z 449.071,A -85,B 0,C 180,E1 -8160.062,E2 -8160.062} C_VEL
LIN {X 0,Y 453.6,Z 451.32,A -85,B 0,C 180,E1 -8160.971,E2 -8160.971} C_VEL
LIN {X 0,Y 452.502,Z 452.711,A -85,B 0,C 180,E1 -8161.686,E2 -8161.686} C_VEL
LIN {X 0,Y 452.404,Z 453.068,A -85,B 0,C 180,E1 -8161.929,E2 -8161.929} C_VEL
LIN {X 0,Y 452.322,Z 454.689,A -85,B 0,C 180,E1 -8163.219,E2 -8163.219} C_VEL
LIN {X 0,Y 452.316,Z 455.399,A -85,B 0,C 180,E1 -8164.316,E2 -8164.316} C_VEL
LIN {X 0,Y 452.288,Z 455.499,A -85,B 0,C 180,E1 -8165.194,E2 -8165.194} C_VEL
LIN {X 0,Y 452.319,Z 455.009,A -85,B 0,C 180,E1 -8166.453,E2 -8166.453} C_VEL
LIN {X 0,Y 452.406,Z 453.106,A -85,B 0,C 180,E1 -8168.11,E2 -8168.11} C_VEL
LIN {X 0,Y 452.592,Z 450.299,A -85,B 0,C 180,E1 -8169.55,E2 -8169.55} C_VEL
LIN {X 0,Y 452.789,Z 445.564,A -85,B 0,C 180,E1 -8171.231,E2 -8171.231} C_VEL
LIN {X 0,Y 452.981,Z 440.297,A -85,B 0,C 180,E1 -8172.623,E2 -8172.623} C_VEL
LIN {X 0,Y 453.353,Z 433.072,A -85,B 0,C 180,E1 -8174.107,E2 -8174.107} C_VEL
LIN {X 0,Y 453.78,Z 425.055,A -85,B 0,C 180,E1 -8175.423,E2 -8175.423} C_VEL
LIN {X 0,Y 454.261,Z 416.388,A -85,B 0,C 180,E1 -8176.581,E2 -8176.581} C_VEL
LIN {X 0,Y 454.778,Z 406.837,A -85,B 0,C 180,E1 -8177.618,E2 -8177.618} C_VEL
LIN {X 0,Y 455.292,Z 396.415,A -85,B 0,C 180,E1 -8178.537,E2 -8178.537} C_VEL
LIN {X 0,Y 455.935,Z 383.933,A -85,B 0,C 180,E1 -8179.402,E2 -8179.402} C_VEL
LIN {X 0,Y 456.335,Z 371.565,A -85,B 0,C 180,E1 -8180.045,E2 -8180.045} C_VEL
LIN {X 0,Y 456.68,Z 359.131,A -85,B 0,C 180,E1 -8180.505,E2 -8180.505} C_VEL
LIN {X 0,Y 456.941,Z 346.257,A -85,B 0,C 180,E1 -8180.805,E2 -8180.805} C_VEL
LIN {X 0,Y 457.619,Z 260.885,A -85,B 0,C 180,E1 -8182.168,E2 -8182.168} C_VEL
LIN {X 0,Y 454.526,Z 244.536,A -85,B 0,C 180,E1 -8182.583,E2 -8182.583} C_VEL
LIN {X 0,Y 454.999,Z 232.377,A -85,B 0,C 180,E1 -8185.127,E2 -8185.127} C_VEL
LIN {X 0,Y 453.692,Z 222.974,A -85,B 0,C 180,E1 -8187.225,E2 -8187.225} C_VEL
LIN {X 0,Y 453.792,Z 222.958,A -85,B 0,C 180,E1 -8190,E2 -8190} C_VEL
LIN {X 0,Y 453.709,Z 222.965,A -85,B 0,C 180,E1 -8192.663,E2 -8192.663} C_VEL
LIN {X 0,Y 453.641,Z 222.975,A -85,B 0,C 180,E1 -8196.226,E2 -8196.226} C_VEL
LIN {X 0,Y 453.586,Z 222.981,A -85,B 0,C 180,E1 -8198.913,E2 -8198.913} C_VEL
LIN {X 0,Y 453.567,Z 222.984,A -85,B 0,C 180,E1 -8202.529,E2 -8202.529} C_VEL
LIN {X 0,Y 453.54,Z 222.988,A -85,B 0,C 180,E1 -8206.196,E2 -8206.196} C_VEL
LIN {X 0,Y 453.519,Z 222.991,A -85,B 0,C 180,E1 -8209.039,E2 -8209.039} C_VEL
LIN {X 0,Y 453.478,Z 222.999,A -85,B 0,C 180,E1 -8211.836,E2 -8211.836} C_VEL
LIN {X 0,Y 453.495,Z 222.994,A -85,B 0,C 180,E1 -8214.735,E2 -8214.735} C_VEL
LIN {X 0,Y 453.508,Z 222.994,A -85,B 0,C 180,E1 -8217.953,E2 -8217.953} C_VEL
LIN {X 0,Y 453.476,Z 222.997,A -85,B 0,C 180,E1 -8220.759,E2 -8220.759} C_VEL
LIN {X 0,Y 453.477,Z 222.998,A -85,B 0,C 180,E1 -8223.912,E2 -8223.912} C_VEL
LIN {X 0,Y 453.45,Z 223.001,A -85,B 0,C 180,E1 -8227.189,E2 -8227.189} C_VEL
LIN {X 0,Y 453.493,Z 222.995,A -85,B 0,C 180,E1 -8230.609,E2 -8230.609} C_VEL
LIN {X 0,Y 453.46,Z 222.999,A -85,B 0,C 180,E1 -8234.221,E2 -8234.221} C_VEL
LIN {X 0,Y 453.46,Z 222.999,A -85,B 0,C 180,E1 -8237.004,E2 -8237.004} C_VEL
LIN {X 0,Y 453.493,Z 222.997,A -85,B 0,C 180,E1 -8239.409,E2 -8239.409} C_VEL
LIN {X 0,Y 453.449,Z 223,A -85,B 0,C 180,E1 -8242.227,E2 -8242.227} C_VEL
LIN {X 0,Y 453.487,Z 222.997,A -85,B 0,C 180,E1 -8245.222,E2 -8245.222} C_VEL
LIN {X 0,Y 453.464,Z 222.999,A -85,B 0,C 180,E1 -8248.474,E2 -8248.474} C_VEL
LIN {X 0,Y 453.53,Z 222.991,A -85,B 0,C 180,E1 -8252.04,E2 -8252.04} C_VEL
LIN {X 0,Y 453.512,Z 222.994,A -85,B 0,C 180,E1 -8255.265,E2 -8255.265} C_VEL
LIN {X 0,Y 453.478,Z 222.997,A -85,B 0,C 180,E1 -8258.415,E2 -8258.415} C_VEL
LIN {X 0,Y 453.519,Z 222.992,A -85,B 0,C 180,E1 -8261.008,E2 -8261.008} C_VEL
LIN {X 0,Y 453.566,Z 222.986,A -85,B 0,C 180,E1 -8263.879,E2 -8263.879} C_VEL
LIN {X 0,Y 453.561,Z 222.988,A -85,B 0,C 180,E1 -8267.471,E2 -8267.471} C_VEL
LIN {X 0,Y 453.59,Z 222.984,A -85,B 0,C 180,E1 -8271.086,E2 -8271.086} C_VEL
LIN {X 0,Y 453.676,Z 222.973,A -85,B 0,C 180,E1 -8273.775,E2 -8273.775} C_VEL
LIN {X 0,Y 453.762,Z 222.962,A -85,B 0,C 180,E1 -8277.337,E2 -8277.337} C_VEL
LIN {X 0,Y 453.82,Z 222.954,A -85,B 0,C 180,E1 -8280,E2 -8280} C_VEL
LIN {X 0,Y 453.762,Z 222.964,A -85,B 0,C 180,E1 -8282.663,E2 -8282.663} C_VEL
LIN {X 0,Y 453.676,Z 222.973,A -85,B 0,C 180,E1 -8286.225,E2 -8286.225} C_VEL
LIN {X 0,Y 453.589,Z 222.984,A -85,B 0,C 180,E1 -8288.913,E2 -8288.913} C_VEL
LIN {X 0,Y 453.56,Z 222.989,A -85,B 0,C 180,E1 -8292.529,E2 -8292.529} C_VEL
LIN {X 0,Y 453.542,Z 222.989,A -85,B 0,C 180,E1 -8296.196,E2 -8296.196} C_VEL
LIN {X 0,Y 453.518,Z 222.992,A -85,B 0,C 180,E1 -8299.041,E2 -8299.041} C_VEL
LIN {X 0,Y 453.474,Z 222.997,A -85,B 0,C 180,E1 -8301.836,E2 -8301.836} C_VEL
LIN {X 0,Y 453.512,Z 222.995,A -85,B 0,C 180,E1 -8304.735,E2 -8304.735} C_VEL
LIN {X 0,Y 453.53,Z 222.99,A -85,B 0,C 180,E1 -8307.96,E2 -8307.96} C_VEL
LIN {X 0,Y 453.463,Z 222.998,A -85,B 0,C 180,E1 -8311.525,E2 -8311.525} C_VEL
LIN {X 0,Y 453.487,Z 222.998,A -85,B 0,C 180,E1 -8314.778,E2 -8314.778} C_VEL
LIN {X 0,Y 453.463,Z 223,A -85,B 0,C 180,E1 -8318.312,E2 -8318.312} C_VEL
LIN {X 0,Y 453.492,Z 222.999,A -85,B 0,C 180,E1 -8320.609,E2 -8320.609} C_VEL
LIN {X 0,Y 453.454,Z 222.999,A -85,B 0,C 180,E1 -8323.245,E2 -8323.245} C_VEL
LIN {X 0,Y 453.465,Z 222.997,A -85,B 0,C 180,E1 -8325.779,E2 -8325.779} C_VEL
LIN {X 0,Y 453.478,Z 222.997,A -85,B 0,C 180,E1 -8328.21,E2 -8328.21} C_VEL
LIN {X 0,Y 453.508,Z 222.994,A -85,B 0,C 180,E1 -8330.791,E2 -8330.791} C_VEL
LIN {X 0,Y 453.451,Z 222.998,A -85,B 0,C 180,E1 -8333.917,E2 -8333.917} C_VEL
LIN {X 0,Y 453.483,Z 222.997,A -85,B 0,C 180,E1 -8337.152,E2 -8337.152} C_VEL
LIN {X 0,Y 453.475,Z 223,A -85,B 0,C 180,E1 -8340.269,E2 -8340.269} C_VEL
LIN {X 0,Y 453.491,Z 223,A -85,B 0,C 180,E1 -8343.293,E2 -8343.293} C_VEL
LIN {X 0,Y 453.534,Z 223.09,A -85,B 0,C 180,E1 -8343.94,E2 -8343.94} C_VEL
LIN {X 0,Y 455.825,Z 235.115,A -85,B 0,C 180,E1 -8346.368,E2 -8346.368} C_VEL
LIN {X 0,Y 455.462,Z 245.256,A -85,B 0,C 180,E1 -8348.264,E2 -8348.264} C_VEL
LIN {X 0,Y 454.584,Z 262.975,A -85,B 0,C 180,E1 -8351.523,E2 -8351.523} C_VEL
LIN {X 0,Y 454.382,Z 268.257,A -85,B 0,C 180,E1 -8352.473,E2 -8352.473} C_VEL
LIN {X 0,Y 457.587,Z 289.399,A -85,B 0,C 180,E1 -8352.94,E2 -8352.94} C_VEL
LIN {X 0,Y 456.747,Z 376.71,A -85,B 0,C 180,E1 -8354.351,E2 -8354.351} C_VEL
LIN {X 0,Y 456.363,Z 390.577,A -85,B 0,C 180,E1 -8354.766,E2 -8354.766} C_VEL
LIN {X 0,Y 455.867,Z 403.013,A -85,B 0,C 180,E1 -8355.321,E2 -8355.321} C_VEL
LIN {X 0,Y 455.315,Z 414.912,A -85,B 0,C 180,E1 -8356.044,E2 -8356.044} C_VEL
LIN {X 0,Y 454.705,Z 427.078,A -85,B 0,C 180,E1 -8357,E2 -8357} C_VEL
LIN {X 0,Y 454.249,Z 436.665,A -85,B 0,C 180,E1 -8357.944,E2 -8357.944} C_VEL
LIN {X 0,Y 453.675,Z 445.922,A -85,B 0,C 180,E1 -8359.061,E2 -8359.061} C_VEL
LIN {X 0,Y 453.213,Z 454.922,A -85,B 0,C 180,E1 -8360.404,E2 -8360.404} C_VEL
LIN {X 0,Y 452.905,Z 462.171,A -85,B 0,C 180,E1 -8361.748,E2 -8361.748} C_VEL
LIN {X 0,Y 452.716,Z 467.063,A -85,B 0,C 180,E1 -8362.866,E2 -8362.866} C_VEL
LIN {X 0,Y 452.558,Z 471.815,A -85,B 0,C 180,E1 -8364.207,E2 -8364.207} C_VEL
LIN {X 0,Y 452.485,Z 475.447,A -85,B 0,C 180,E1 -8365.546,E2 -8365.546} C_VEL
LIN {X 0,Y 452.48,Z 477.323,A -85,B 0,C 180,E1 -8366.438,E2 -8366.438} C_VEL
LIN {X 0,Y 452.508,Z 478.731,A -85,B 0,C 180,E1 -8367.33,E2 -8367.33} C_VEL
LIN {X 0,Y 452.429,Z 480.34,A -85,B 0,C 180,E1 -8369.11,E2 -8369.11} C_VEL
LIN {X 0,Y 452.436,Z 480.56,A -85,B 0,C 180,E1 -8370,E2 -8370} C_VEL
LIN {X 0,Y 452.429,Z 480.346,A -85,B 0,C 180,E1 -8370.89,E2 -8370.89} C_VEL
LIN {X 0,Y 452.508,Z 478.738,A -85,B 0,C 180,E1 -8372.671,E2 -8372.671} C_VEL
LIN {X 0,Y 452.479,Z 477.336,A -85,B 0,C 180,E1 -8373.562,E2 -8373.562} C_VEL
LIN {X 0,Y 452.544,Z 474.39,A -85,B 0,C 180,E1 -8374.9,E2 -8374.9} C_VEL
LIN {X 0,Y 452.611,Z 469.866,A -85,B 0,C 180,E1 -8376.396,E2 -8376.396} C_VEL
LIN {X 0,Y 452.81,Z 464.276,A -85,B 0,C 180,E1 -8377.805,E2 -8377.805} C_VEL
LIN {X 0,Y 453.1,Z 457.58,A -85,B 0,C 180,E1 -8379.148,E2 -8379.148} C_VEL
LIN {X 0,Y 453.486,Z 449.273,A -85,B 0,C 180,E1 -8380.492,E2 -8380.492} C_VEL
LIN {X 0,Y 454.038,Z 440.764,A -85,B 0,C 180,E1 -8381.609,E2 -8381.609} C_VEL
LIN {X 0,Y 454.604,Z 431.058,A -85,B 0,C 180,E1 -8382.649,E2 -8382.649} C_VEL
LIN {X 0,Y 455.088,Z 419.849,A -85,B 0,C 180,E1 -8383.622,E2 -8383.622} C_VEL
LIN {X 0,Y 455.673,Z 408.461,A -85,B 0,C 180,E1 -8384.401,E2 -8384.401} C_VEL
LIN {X 0,Y 456.166,Z 396.77,A -85,B 0,C 180,E1 -8385.012,E2 -8385.012} C_VEL
LIN {X 0,Y 456.675,Z 383.326,A -85,B 0,C 180,E1 -8385.509,E2 -8385.509} C_VEL
LIN {X 0,Y 457.003,Z 370.053,A -85,B 0,C 180,E1 -8385.812,E2 -8385.812} C_VEL
LIN {X 0,Y 457.56,Z 287.567,A -85,B 0,C 180,E1 -8387.136,E2 -8387.136} C_VEL
LIN {X 0,Y 454.394,Z 267.707,A -85,B 0,C 180,E1 -8387.6,E2 -8387.6} C_VEL
LIN {X 0,Y 455.094,Z 251.311,A -85,B 0,C 180,E1 -8390.569,E2 -8390.569} C_VEL
LIN {X 0,Y 455.835,Z 235.909,A -85,B 0,C 180,E1 -8393.391,E2 -8393.391} C_VEL
LIN {X 0,Y 454.274,Z 226.859,A -85,B 0,C 180,E1 -8395.179,E2 -8395.179} C_VEL
LIN {X 0,Y 453.514,Z 222.995,A -85,B 0,C 180,E1 -8395.997,E2 -8395.997} C_VEL
LIN {X 0,Y 453.509,Z 222.994,A -85,B 0,C 180,E1 -8398.712,E2 -8398.712} C_VEL
LIN {X 0,Y 453.465,Z 223.002,A -85,B 0,C 180,E1 -8401.799,E2 -8401.799} C_VEL
LIN {X 0,Y 453.48,Z 222.999,A -85,B 0,C 180,E1 -8404.989,E2 -8404.989} C_VEL
LIN {X 0,Y 453.462,Z 222.996,A -85,B 0,C 180,E1 -8408.312,E2 -8408.312} C_VEL
LIN {X 0,Y 453.494,Z 222.992,A -85,B 0,C 180,E1 -8410.609,E2 -8410.609} C_VEL
LIN {X 0,Y 453.472,Z 222.996,A -85,B 0,C 180,E1 -8414.22,E2 -8414.22} C_VEL
LIN {X 0,Y 453.464,Z 223.002,A -85,B 0,C 180,E1 -8417.005,E2 -8417.005} C_VEL
LIN {X 0,Y 453.494,Z 222.998,A -85,B 0,C 180,E1 -8419.409,E2 -8419.409} C_VEL
LIN {X 0,Y 453.45,Z 222.997,A -85,B 0,C 180,E1 -8422.227,E2 -8422.227} C_VEL
LIN {X 0,Y 453.489,Z 222.996,A -85,B 0,C 180,E1 -8425.222,E2 -8425.222} C_VEL
LIN {X 0,Y 453.465,Z 222.994,A -85,B 0,C 180,E1 -8428.475,E2 -8428.475} C_VEL
LIN {X 0,Y 453.532,Z 222.985,A -85,B 0,C 180,E1 -8432.04,E2 -8432.04} C_VEL
LIN {X 0,Y 453.513,Z 222.993,A -85,B 0,C 180,E1 -8435.265,E2 -8435.265} C_VEL
LIN {X 0,Y 453.479,Z 222.994,A -85,B 0,C 180,E1 -8438.415,E2 -8438.415} C_VEL
LIN {X 0,Y 453.521,Z 222.99,A -85,B 0,C 180,E1 -8441.009,E2 -8441.009} C_VEL
LIN {X 0,Y 453.568,Z 222.983,A -85,B 0,C 180,E1 -8443.88,E2 -8443.88} C_VEL
LIN {X 0,Y 453.563,Z 222.985,A -85,B 0,C 180,E1 -8447.471,E2 -8447.471} C_VEL
LIN {X 0,Y 453.591,Z 222.982,A -85,B 0,C 180,E1 -8451.087,E2 -8451.087} C_VEL
LIN {X 0,Y 453.668,Z 222.969,A -85,B 0,C 180,E1 -8453.775,E2 -8453.775} C_VEL
LIN {X 0,Y 453.764,Z 222.961,A -85,B 0,C 180,E1 -8457.337,E2 -8457.337} C_VEL
LIN {X 0,Y 453.822,Z 222.947,A -85,B 0,C 180,E1 -8460,E2 -8460} C_VEL
LIN {X 0,Y 453.763,Z 222.965,A -85,B 0,C 180,E1 -8462.663,E2 -8462.663} C_VEL
LIN {X 0,Y 453.668,Z 222.972,A -85,B 0,C 180,E1 -8466.226,E2 -8466.226} C_VEL
LIN {X 0,Y 453.591,Z 222.985,A -85,B 0,C 180,E1 -8468.913,E2 -8468.913} C_VEL
LIN {X 0,Y 453.563,Z 222.985,A -85,B 0,C 180,E1 -8472.529,E2 -8472.529} C_VEL
LIN {X 0,Y 453.544,Z 222.987,A -85,B 0,C 180,E1 -8476.196,E2 -8476.196} C_VEL
LIN {X 0,Y 453.52,Z 222.993,A -85,B 0,C 180,E1 -8479.041,E2 -8479.041} C_VEL
LIN {X 0,Y 453.476,Z 222.995,A -85,B 0,C 180,E1 -8481.836,E2 -8481.836} C_VEL
LIN {X 0,Y 453.501,Z 222.998,A -85,B 0,C 180,E1 -8484.735,E2 -8484.735} C_VEL
LIN {X 0,Y 453.506,Z 222.993,A -85,B 0,C 180,E1 -8487.954,E2 -8487.954} C_VEL
LIN {X 0,Y 453.475,Z 223,A -85,B 0,C 180,E1 -8490.76,E2 -8490.76} C_VEL
LIN {X 0,Y 453.467,Z 223,A -85,B 0,C 180,E1 -8493.914,E2 -8493.914} C_VEL
LIN {X 0,Y 453.439,Z 223.002,A -85,B 0,C 180,E1 -8497.191,E2 -8497.191} C_VEL
LIN {X 0,Y 453.47,Z 223.001,A -85,B 0,C 180,E1 -8500.612,E2 -8500.612} C_VEL
LIN {X 0,Y 453.495,Z 223.118,A -85,B 0,C 180,E1 -8503.128,E2 -8503.128} C_VEL
LIN {X 0,Y 454.998,Z 231.662,A -85,B 0,C 180,E1 -8504.923,E2 -8504.923} C_VEL
LIN {X 0,Y 454.575,Z 244.478,A -85,B 0,C 180,E1 -8507.46,E2 -8507.46} C_VEL
LIN {X 0,Y 457.893,Z 261.991,A -85,B 0,C 180,E1 -8507.895,E2 -8507.895} C_VEL
LIN {X 0,Y 456.912,Z 352.444,A -85,B 0,C 180,E1 -8509.36,E2 -8509.36} C_VEL
LIN {X 0,Y 456.618,Z 365.521,A -85,B 0,C 180,E1 -8509.752,E2 -8509.752} C_VEL
LIN {X 0,Y 456.231,Z 377.741,A -85,B 0,C 180,E1 -8510.292,E2 -8510.292} C_VEL
LIN {X 0,Y 455.792,Z 388.571,A -85,B 0,C 180,E1 -8510.93,E2 -8510.93} C_VEL
LIN {X 0,Y 455.268,Z 399.194,A -85,B 0,C 180,E1 -8511.727,E2 -8511.727} C_VEL
LIN {X 0,Y 454.661,Z 410.41,A -85,B 0,C 180,E1 -8512.787,E2 -8512.787} C_VEL
LIN {X 0,Y 454.089,Z 420.494,A -85,B 0,C 180,E1 -8513.976,E2 -8513.976} C_VEL
LIN {X 0,Y 453.63,Z 428.817,A -85,B 0,C 180,E1 -8515.197,E2 -8515.197} C_VEL
LIN {X 0,Y 453.236,Z 436.126,A -85,B 0,C 180,E1 -8516.518,E2 -8516.518} C_VEL
LIN {X 0,Y 452.943,Z 442.247,A -85,B 0,C 180,E1 -8517.898,E2 -8517.898} C_VEL
LIN {X 0,Y 452.749,Z 446.765,A -85,B 0,C 180,E1 -8519.186,E2 -8519.186} C_VEL
LIN {X 0,Y 452.611,Z 450.106,A -85,B 0,C 180,E1 -8520.407,E2 -8520.407} C_VEL
LIN {X 0,Y 452.404,Z 453.068,A -85,B 0,C 180,E1 -8521.929,E2 -8521.929} C_VEL
LIN {X 0,Y 451.697,Z 454.18,A -85,B 0,C 180,E1 -8522.66,E2 -8522.66} C_VEL
LIN {X 0,Y 448.773,Z 455.4,A -85,B 0,C 180,E1 -8523.857,E2 -8523.857} C_VEL
LIN {X 0,Y 446.322,Z 455.766,A -85,B 0,C 180,E1 -8524.83,E2 -8524.83} C_VEL
LIN {X 0,Y 445.276,Z 455.659,A -85,B 0,C 180,E1 -8525.582,E2 -8525.582} C_VEL
LIN {X 0,Y 445.194,Z 455.545,A -85,B 0,C 180,E1 -8525.836,E2 -8525.836} C_VEL
LIN {X 0,Y 445.216,Z 454.96,A -85,B 0,C 180,E1 -8526.757,E2 -8526.757} C_VEL
LIN {X 0,Y 445.284,Z 453.895,A -85,B 0,C 180,E1 -8527.741,E2 -8527.741} C_VEL
LIN {X 0,Y 445.456,Z 451.401,A -85,B 0,C 180,E1 -8529.208,E2 -8529.208} C_VEL
LIN {X 0,Y 445.642,Z 447.808,A -85,B 0,C 180,E1 -8530.66,E2 -8530.66} C_VEL
LIN {X 0,Y 445.807,Z 443.045,A -85,B 0,C 180,E1 -8532.097,E2 -8532.097} C_VEL
LIN {X 0,Y 446.096,Z 436.927,A -85,B 0,C 180,E1 -8533.526,E2 -8533.526} C_VEL
LIN {X 0,Y 446.549,Z 429.256,A -85,B 0,C 180,E1 -8534.949,E2 -8534.949} C_VEL
LIN {X 0,Y 446.996,Z 421.429,A -85,B 0,C 180,E1 -8536.127,E2 -8536.127} C_VEL
LIN {X 0,Y 447.573,Z 411.886,A -85,B 0,C 180,E1 -8537.301,E2 -8537.301} C_VEL
LIN {X 0,Y 448.173,Z 401.207,A -85,B 0,C 180,E1 -8538.352,E2 -8538.352} C_VEL
LIN {X 0,Y 448.824,Z 389.286,A -85,B 0,C 180,E1 -8539.284,E2 -8539.284} C_VEL
LIN {X 0,Y 449.269,Z 377.789,A -85,B 0,C 180,E1 -8539.978,E2 -8539.978} C_VEL
LIN {X 0,Y 449.681,Z 364.498,A -85,B 0,C 180,E1 -8540.565,E2 -8540.565} C_VEL
LIN {X 0,Y 449.975,Z 351.754,A -85,B 0,C 180,E1 -8540.941,E2 -8540.941} C_VEL
LIN {X 0,Y 450.855,Z 261.788,A -85,B 0,C 180,E1 -8542.414,E2 -8542.414} C_VEL
LIN {X 0,Y 447.593,Z 244.785,A -85,B 0,C 180,E1 -8542.84,E2 -8542.84} C_VEL
LIN {X 0,Y 448.027,Z 233.304,A -85,B 0,C 180,E1 -8545.276,E2 -8545.276} C_VEL
LIN {X 0,Y 446.673,Z 223.849,A -85,B 0,C 180,E1 -8547.407,E2 -8547.407} C_VEL
LIN {X 0,Y 446.741,Z 223.836,A -85,B 0,C 180,E1 -8550,E2 -8550} C_VEL
LIN {X 0,Y 446.658,Z 223.843,A -85,B 0,C 180,E1 -8552.705,E2 -8552.705} C_VEL
LIN {X 0,Y 446.611,Z 223.85,A -85,B 0,C 180,E1 -8556.324,E2 -8556.324} C_VEL
LIN {X 0,Y 446.534,Z 223.86,A -85,B 0,C 180,E1 -8559.055,E2 -8559.055} C_VEL
LIN {X 0,Y 446.524,Z 223.861,A -85,B 0,C 180,E1 -8562.729,E2 -8562.729} C_VEL
LIN {X 0,Y 446.487,Z 223.866,A -85,B 0,C 180,E1 -8566.459,E2 -8566.459} C_VEL
LIN {X 0,Y 446.47,Z 223.87,A -85,B 0,C 180,E1 -8569.303,E2 -8569.303} C_VEL
LIN {X 0,Y 446.419,Z 223.875,A -85,B 0,C 180,E1 -8572.199,E2 -8572.199} C_VEL
LIN {X 0,Y 446.44,Z 223.873,A -85,B 0,C 180,E1 -8575.153,E2 -8575.153} C_VEL
LIN {X 0,Y 446.45,Z 223.872,A -85,B 0,C 180,E1 -8578.181,E2 -8578.181} C_VEL
LIN {X 0,Y 446.416,Z 223.877,A -85,B 0,C 180,E1 -8581.3,E2 -8581.3} C_VEL
LIN {X 0,Y 446.429,Z 223.874,A -85,B 0,C 180,E1 -8584.523,E2 -8584.523} C_VEL
LIN {X 0,Y 446.411,Z 223.877,A -85,B 0,C 180,E1 -8588.078,E2 -8588.078} C_VEL
LIN {X 0,Y 446.422,Z 223.876,A -85,B 0,C 180,E1 -8590.916,E2 -8590.916} C_VEL
LIN {X 0,Y 446.398,Z 223.881,A -85,B 0,C 180,E1 -8593.846,E2 -8593.846} C_VEL
LIN {X 0,Y 446.395,Z 223.879,A -85,B 0,C 180,E1 -8596.403,E2 -8596.403} C_VEL
LIN {X 0,Y 446.426,Z 223.875,A -85,B 0,C 180,E1 -8599.082,E2 -8599.082} C_VEL
LIN {X 0,Y 446.408,Z 223.878,A -85,B 0,C 180,E1 -8602.121,E2 -8602.121} C_VEL
LIN {X 0,Y 446.429,Z 223.877,A -85,B 0,C 180,E1 -8605.477,E2 -8605.477} C_VEL
LIN {X 0,Y 446.414,Z 223.878,A -85,B 0,C 180,E1 -8608.699,E2 -8608.699} C_VEL
LIN {X 0,Y 446.483,Z 223.87,A -85,B 0,C 180,E1 -8611.821,E2 -8611.821} C_VEL
LIN {X 0,Y 446.456,Z 223.872,A -85,B 0,C 180,E1 -8614.847,E2 -8614.847} C_VEL
LIN {X 0,Y 446.446,Z 223.873,A -85,B 0,C 180,E1 -8618.245,E2 -8618.245} C_VEL
LIN {X 0,Y 446.454,Z 223.874,A -85,B 0,C 180,E1 -8621.649,E2 -8621.649} C_VEL
LIN {X 0,Y 446.505,Z 223.867,A -85,B 0,C 180,E1 -8624.48,E2 -8624.48} C_VEL
LIN {X 0,Y 446.515,Z 223.865,A -85,B 0,C 180,E1 -8628.193,E2 -8628.193} C_VEL
LIN {X 0,Y 446.598,Z 223.855,A -85,B 0,C 180,E1 -8631.858,E2 -8631.858} C_VEL
LIN {X 0,Y 446.644,Z 223.851,A -85,B 0,C 180,E1 -8634.582,E2 -8634.582} C_VEL
LIN {X 0,Y 446.706,Z 223.841,A -85,B 0,C 180,E1 -8637.295,E2 -8637.295} C_VEL
LIN {X 0,Y 446.79,Z 223.83,A -85,B 0,C 180,E1 -8640,E2 -8640} C_VEL
LIN {X 0,Y 446.706,Z 223.843,A -85,B 0,C 180,E1 -8642.705,E2 -8642.705} C_VEL
LIN {X 0,Y 446.645,Z 223.849,A -85,B 0,C 180,E1 -8646.324,E2 -8646.324} C_VEL
LIN {X 0,Y 446.535,Z 223.862,A -85,B 0,C 180,E1 -8649.055,E2 -8649.055} C_VEL
LIN {X 0,Y 446.518,Z 223.866,A -85,B 0,C 180,E1 -8652.73,E2 -8652.73} C_VEL
LIN {X 0,Y 446.493,Z 223.868,A -85,B 0,C 180,E1 -8656.228,E2 -8656.228} C_VEL
LIN {X 0,Y 446.467,Z 223.87,A -85,B 0,C 180,E1 -8659.303,E2 -8659.303} C_VEL
LIN {X 0,Y 446.416,Z 223.877,A -85,B 0,C 180,E1 -8662.2,E2 -8662.2} C_VEL
LIN {X 0,Y 446.455,Z 223.871,A -85,B 0,C 180,E1 -8665.152,E2 -8665.152} C_VEL
LIN {X 0,Y 446.482,Z 223.869,A -85,B 0,C 180,E1 -8668.179,E2 -8668.179} C_VEL
LIN {X 0,Y 446.417,Z 223.876,A -85,B 0,C 180,E1 -8671.775,E2 -8671.775} C_VEL
LIN {X 0,Y 446.429,Z 223.879,A -85,B 0,C 180,E1 -8674.523,E2 -8674.523} C_VEL
LIN {X 0,Y 446.414,Z 223.876,A -85,B 0,C 180,E1 -8678.08,E2 -8678.08} C_VEL
LIN {X 0,Y 446.425,Z 223.876,A -85,B 0,C 180,E1 -8680.918,E2 -8680.918} C_VEL
LIN {X 0,Y 446.4,Z 223.877,A -85,B 0,C 180,E1 -8683.846,E2 -8683.846} C_VEL
LIN {X 0,Y 446.399,Z 223.881,A -85,B 0,C 180,E1 -8686.404,E2 -8686.404} C_VEL
LIN {X 0,Y 446.426,Z 223.874,A -85,B 0,C 180,E1 -8689.083,E2 -8689.083} C_VEL
LIN {X 0,Y 446.413,Z 223.875,A -85,B 0,C 180,E1 -8691.921,E2 -8691.921} C_VEL
LIN {X 0,Y 446.428,Z 223.873,A -85,B 0,C 180,E1 -8695.477,E2 -8695.477} C_VEL
LIN {X 0,Y 446.416,Z 223.88,A -85,B 0,C 180,E1 -8698.7,E2 -8698.7} C_VEL
LIN {X 0,Y 446.485,Z 223.869,A -85,B 0,C 180,E1 -8701.822,E2 -8701.822} C_VEL
LIN {X 0,Y 446.488,Z 223.924,A -85,B 0,C 180,E1 -8703.708,E2 -8703.708} C_VEL
LIN {X 0,Y 448.843,Z 236.154,A -85,B 0,C 180,E1 -8706.222,E2 -8706.222} C_VEL
LIN {X 0,Y 448.713,Z 241.881,A -85,B 0,C 180,E1 -8707.317,E2 -8707.317} C_VEL
LIN {X 0,Y 447.894,Z 258.46,A -85,B 0,C 180,E1 -8710.43,E2 -8710.43} C_VEL
LIN {X 0,Y 447.415,Z 267.985,A -85,B 0,C 180,E1 -8712.197,E2 -8712.197} C_VEL
LIN {X 0,Y 450.782,Z 289.373,A -85,B 0,C 180,E1 -8712.684,E2 -8712.684} C_VEL
LIN {X 0,Y 449.921,Z 376.198,A -85,B 0,C 180,E1 -8714.107,E2 -8714.107} C_VEL
LIN {X 0,Y 449.536,Z 389.41,A -85,B 0,C 180,E1 -8714.5,E2 -8714.5} C_VEL
LIN {X 0,Y 449.058,Z 401.558,A -85,B 0,C 180,E1 -8715.035,E2 -8715.035} C_VEL
LIN {X 0,Y 448.487,Z 413.013,A -85,B 0,C 180,E1 -8715.711,E2 -8715.711} C_VEL
LIN {X 0,Y 447.872,Z 424.948,A -85,B 0,C 180,E1 -8716.632,E2 -8716.632} C_VEL
LIN {X 0,Y 447.328,Z 435.342,A -85,B 0,C 180,E1 -8717.64,E2 -8717.64} C_VEL
LIN {X 0,Y 446.831,Z 443.971,A -85,B 0,C 180,E1 -8718.662,E2 -8718.662} C_VEL
LIN {X 0,Y 446.335,Z 451.923,A -85,B 0,C 180,E1 -8719.797,E2 -8719.797} C_VEL
LIN {X 0,Y 445.962,Z 459.701,A -85,B 0,C 180,E1 -8721.162,E2 -8721.162} C_VEL
LIN {X 0,Y 445.633,Z 466.844,A -85,B 0,C 180,E1 -8722.752,E2 -8722.752} C_VEL
LIN {X 0,Y 445.482,Z 471.05,A -85,B 0,C 180,E1 -8723.94,E2 -8723.94} C_VEL
LIN {X 0,Y 445.411,Z 475.24,A -85,B 0,C 180,E1 -8725.475,E2 -8725.475} C_VEL
LIN {X 0,Y 445.378,Z 477.117,A -85,B 0,C 180,E1 -8726.381,E2 -8726.381} C_VEL
LIN {X 0,Y 445.432,Z 478.529,A -85,B 0,C 180,E1 -8727.287,E2 -8727.287} C_VEL
LIN {X 0,Y 445.339,Z 480.142,A -85,B 0,C 180,E1 -8729.096,E2 -8729.096} C_VEL
LIN {X 0,Y 445.343,Z 480.364,A -85,B 0,C 180,E1 -8730,E2 -8730} C_VEL
LIN {X 0,Y 445.339,Z 480.151,A -85,B 0,C 180,E1 -8730.904,E2 -8730.904} C_VEL
LIN {X 0,Y 445.432,Z 478.545,A -85,B 0,C 180,E1 -8732.713,E2 -8732.713} C_VEL
LIN {X 0,Y 445.378,Z 477.144,A -85,B 0,C 180,E1 -8733.619,E2 -8733.619} C_VEL
LIN {X 0,Y 445.473,Z 474.2,A -85,B 0,C 180,E1 -8734.978,E2 -8734.978} C_VEL
LIN {X 0,Y 445.559,Z 468.78,A -85,B 0,C 180,E1 -8736.749,E2 -8736.749} C_VEL
LIN {X 0,Y 445.787,Z 463.072,A -85,B 0,C 180,E1 -8738.157,E2 -8738.157} C_VEL
LIN {X 0,Y 446.13,Z 456.155,A -85,B 0,C 180,E1 -8739.521,E2 -8739.521} C_VEL
LIN {X 0,Y 446.579,Z 447.508,A -85,B 0,C 180,E1 -8740.886,E2 -8740.886} C_VEL
LIN {X 0,Y 447.163,Z 438.645,A -85,B 0,C 180,E1 -8742.02,E2 -8742.02} C_VEL
LIN {X 0,Y 447.801,Z 427.887,A -85,B 0,C 180,E1 -8743.14,E2 -8743.14} C_VEL
LIN {X 0,Y 448.34,Z 416.748,A -85,B 0,C 180,E1 -8744.062,E2 -8744.062} C_VEL
LIN {X 0,Y 448.966,Z 404.436,A -85,B 0,C 180,E1 -8744.852,E2 -8744.852} C_VEL
LIN {X 0,Y 449.532,Z 392.803,A -85,B 0,C 180,E1 -8745.413,E2 -8745.413} C_VEL
LIN {X 0,Y 449.904,Z 380.492,A -85,B 0,C 180,E1 -8745.836,E2 -8745.836} C_VEL
LIN {X 0,Y 450.247,Z 364.953,A -85,B 0,C 180,E1 -8746.143,E2 -8746.143} C_VEL
LIN {X 0,Y 450.765,Z 288.008,A -85,B 0,C 180,E1 -8747.399,E2 -8747.399} C_VEL
LIN {X 0,Y 447.446,Z 267.459,A -85,B 0,C 180,E1 -8747.899,E2 -8747.899} C_VEL
LIN {X 0,Y 448.201,Z 251.143,A -85,B 0,C 180,E1 -8750.9,E2 -8750.9} C_VEL
LIN {X 0,Y 448.89,Z 237.02,A -85,B 0,C 180,E1 -8753.531,E2 -8753.531} C_VEL
LIN {X 0,Y 447.033,Z 226.673,A -85,B 0,C 180,E1 -8755.616,E2 -8755.616} C_VEL
LIN {X 0,Y 446.457,Z 223.874,A -85,B 0,C 180,E1 -8756.197,E2 -8756.197} C_VEL
LIN {X 0,Y 446.448,Z 223.874,A -85,B 0,C 180,E1 -8759.209,E2 -8759.209} C_VEL
LIN {X 0,Y 446.423,Z 223.877,A -85,B 0,C 180,E1 -8762.361,E2 -8762.361} C_VEL
LIN {X 0,Y 446.418,Z 223.878,A -85,B 0,C 180,E1 -8765.626,E2 -8765.626} C_VEL
LIN {X 0,Y 446.441,Z 223.875,A -85,B 0,C 180,E1 -8769.027,E2 -8769.027} C_VEL
LIN {X 0,Y 446.436,Z 223.871,A -85,B 0,C 180,E1 -8772.277,E2 -8772.277} C_VEL
LIN {X 0,Y 446.455,Z 223.874,A -85,B 0,C 180,E1 -8775.103,E2 -8775.103} C_VEL
LIN {X 0,Y 446.428,Z 223.871,A -85,B 0,C 180,E1 -8778.609,E2 -8778.609} C_VEL
LIN {X 0,Y 446.441,Z 223.875,A -85,B 0,C 180,E1 -8780.973,E2 -8780.973} C_VEL
LIN {X 0,Y 446.421,Z 223.872,A -85,B 0,C 180,E1 -8784.374,E2 -8784.374} C_VEL
LIN {X 0,Y 446.422,Z 223.872,A -85,B 0,C 180,E1 -8787.638,E2 -8787.638} C_VEL
LIN {X 0,Y 446.448,Z 223.873,A -85,B 0,C 180,E1 -8790.791,E2 -8790.791} C_VEL
LIN {X 0,Y 446.477,Z 223.866,A -85,B 0,C 180,E1 -8793.848,E2 -8793.848} C_VEL
LIN {X 0,Y 446.428,Z 223.874,A -85,B 0,C 180,E1 -8796.823,E2 -8796.823} C_VEL
LIN {X 0,Y 446.443,Z 223.87,A -85,B 0,C 180,E1 -8799.737,E2 -8799.737} C_VEL
LIN {X 0,Y 446.461,Z 223.868,A -85,B 0,C 180,E1 -8802.597,E2 -8802.597} C_VEL
LIN {X 0,Y 446.47,Z 223.863,A -85,B 0,C 180,E1 -8805.412,E2 -8805.412} C_VEL
LIN {X 0,Y 446.517,Z 223.861,A -85,B 0,C 180,E1 -8808.193,E2 -8808.193} C_VEL
LIN {X 0,Y 446.6,Z 223.85,A -85,B 0,C 180,E1 -8811.858,E2 -8811.858} C_VEL
LIN {X 0,Y 446.641,Z 223.849,A -85,B 0,C 180,E1 -8814.583,E2 -8814.583} C_VEL
LIN {X 0,Y 446.708,Z 223.84,A -85,B 0,C 180,E1 -8817.295,E2 -8817.295} C_VEL
LIN {X 0,Y 446.792,Z 223.822,A -85,B 0,C 180,E1 -8820,E2 -8820} C_VEL
LIN {X 0,Y 446.707,Z 223.843,A -85,B 0,C 180,E1 -8822.705,E2 -8822.705} C_VEL
LIN {X 0,Y 446.638,Z 223.849,A -85,B 0,C 180,E1 -8826.324,E2 -8826.324} C_VEL
LIN {X 0,Y 446.537,Z 223.863,A -85,B 0,C 180,E1 -8829.055,E2 -8829.055} C_VEL
LIN {X 0,Y 446.521,Z 223.865,A -85,B 0,C 180,E1 -8832.73,E2 -8832.73} C_VEL
LIN {X 0,Y 446.496,Z 223.865,A -85,B 0,C 180,E1 -8836.228,E2 -8836.228} C_VEL
LIN {X 0,Y 446.469,Z 223.869,A -85,B 0,C 180,E1 -8839.303,E2 -8839.303} C_VEL
LIN {X 0,Y 446.418,Z 223.876,A -85,B 0,C 180,E1 -8842.2,E2 -8842.2} C_VEL
LIN {X 0,Y 446.443,Z 223.873,A -85,B 0,C 180,E1 -8845.153,E2 -8845.153} C_VEL
LIN {X 0,Y 446.449,Z 223.874,A -85,B 0,C 180,E1 -8848.181,E2 -8848.181} C_VEL
LIN {X 0,Y 446.415,Z 223.875,A -85,B 0,C 180,E1 -8851.301,E2 -8851.301} C_VEL
LIN {X 0,Y 446.422,Z 223.879,A -85,B 0,C 180,E1 -8854.524,E2 -8854.524} C_VEL
LIN {X 0,Y 446.402,Z 223.882,A -85,B 0,C 180,E1 -8858.077,E2 -8858.077} C_VEL
LIN {X 0,Y 446.406,Z 223.879,A -85,B 0,C 180,E1 -8861.394,E2 -8861.394} C_VEL
LIN {X 0,Y 446.446,Z 223.99,A -85,B 0,C 180,E1 -8862.91,E2 -8862.91} C_VEL
LIN {X 0,Y 447.948,Z 231.871,A -85,B 0,C 180,E1 -8864.596,E2 -8864.596} C_VEL
LIN {X 0,Y 447.71,Z 242.137,A -85,B 0,C 180,E1 -8866.657,E2 -8866.657} C_VEL
LIN {X 0,Y 447.657,Z 244.773,A -85,B 0,C 180,E1 -8867.182,E2 -8867.182} C_VEL
LIN {X 0,Y 451.079,Z 262.099,A -85,B 0,C 180,E1 -8867.618,E2 -8867.618} C_VEL
LIN {X 0,Y 450.128,Z 352.095,A -85,B 0,C 180,E1 -8869.097,E2 -8869.097} C_VEL
LIN {X 0,Y 449.81,Z 365.63,A -85,B 0,C 180,E1 -8869.505,E2 -8869.505} C_VEL
LIN {X 0,Y 449.391,Z 377.312,A -85,B 0,C 180,E1 -8870.024,E2 -8870.024} C_VEL
LIN {X 0,Y 448.905,Z 389.043,A -85,B 0,C 180,E1 -8870.722,E2 -8870.722} C_VEL
LIN {X 0,Y 448.294,Z 400.574,A -85,B 0,C 180,E1 -8871.616,E2 -8871.616} C_VEL
LIN {X 0,Y 447.677,Z 411.357,A -85,B 0,C 180,E1 -8872.667,E2 -8872.667} C_VEL
LIN {X 0,Y 447.154,Z 420.326,A -85,B 0,C 180,E1 -8873.747,E2 -8873.747} C_VEL
LIN {X 0,Y 446.699,Z 428.19,A -85,B 0,C 180,E1 -8874.898,E2 -8874.898} C_VEL
LIN {X 0,Y 446.239,Z 435.835,A -85,B 0,C 180,E1 -8876.278,E2 -8876.278} C_VEL
LIN {X 0,Y 445.913,Z 441.723,A -85,B 0,C 180,E1 -8877.597,E2 -8877.597} C_VEL
LIN {X 0,Y 445.67,Z 447.214,A -85,B 0,C 180,E1 -8879.169,E2 -8879.169} C_VEL
LIN {X 0,Y 445.485,Z 451.21,A -85,B 0,C 180,E1 -8880.721,E2 -8880.721} C_VEL
LIN {X 0,Y 445.302,Z 453.671,A -85,B 0,C 180,E1 -8882.108,E2 -8882.108} C_VEL
LIN {X 0,Y 445.221,Z 455.326,A -85,B 0,C 180,E1 -8883.769,E2 -8883.769} C_VEL
LIN {X 0,Y 445.196,Z 455.682,A -85,B 0,C 180,E1 -8884.771,E2 -8884.771} C_VEL
LIN {X 0,Y 445.194,Z 455.545,A -85,B 0,C 180,E1 -8885.836,E2 -8885.836} C_VEL
LIN {X 0,Y 444.545,Z 455.128,A -85,B 0,C 180,E1 -8886.59,E2 -8886.59} C_VEL
LIN {X 0,Y 441.755,Z 453.928,A -85,B 0,C 180,E1 -8887.812,E2 -8887.812} C_VEL
LIN {X 0,Y 439.43,Z 452.483,A -85,B 0,C 180,E1 -8888.786,E2 -8888.786} C_VEL
LIN {X 0,Y 438.481,Z 451.041,A -85,B 0,C 180,E1 -8889.529,E2 -8889.529} C_VEL
LIN {X 0,Y 438.431,Z 450.466,A -85,B 0,C 180,E1 -8889.778,E2 -8889.778} C_VEL
LIN {X 0,Y 438.632,Z 446.284,A -85,B 0,C 180,E1 -8891.31,E2 -8891.31} C_VEL
LIN {X 0,Y 438.84,Z 441.034,A -85,B 0,C 180,E1 -8892.766,E2 -8892.766} C_VEL
LIN {X 0,Y 439.23,Z 434.353,A -85,B 0,C 180,E1 -8894.216,E2 -8894.216} C_VEL
LIN {X 0,Y 439.733,Z 425.982,A -85,B 0,C 180,E1 -8895.657,E2 -8895.657} C_VEL
LIN {X 0,Y 440.337,Z 416.499,A -85,B 0,C 180,E1 -8896.968,E2 -8896.968} C_VEL
LIN {X 0,Y 440.894,Z 406.846,A -85,B 0,C 180,E1 -8898.04,E2 -8898.04} C_VEL
LIN {X 0,Y 441.518,Z 396.297,A -85,B 0,C 180,E1 -8898.988,E2 -8898.988} C_VEL
LIN {X 0,Y 442.166,Z 384.687,A -85,B 0,C 180,E1 -8899.815,E2 -8899.815} C_VEL
LIN {X 0,Y 442.582,Z 373.227,A -85,B 0,C 180,E1 -8900.445,E2 -8900.445} C_VEL
LIN {X 0,Y 442.953,Z 361.021,A -85,B 0,C 180,E1 -8900.928,E2 -8900.928} C_VEL
LIN {X 0,Y 443.216,Z 348.496,A -85,B 0,C 180,E1 -8901.25,E2 -8901.25} C_VEL
LIN {X 0,Y 444.059,Z 262.603,A -85,B 0,C 180,E1 -8902.669,E2 -8902.669} C_VEL
LIN {X 0,Y 440.684,Z 244.912,A -85,B 0,C 180,E1 -8903.13,E2 -8903.13} C_VEL
LIN {X 0,Y 441.046,Z 234.237,A -85,B 0,C 180,E1 -8905.43,E2 -8905.43} C_VEL
LIN {X 0,Y 439.62,Z 224.727,A -85,B 0,C 180,E1 -8907.652,E2 -8907.652} C_VEL
LIN {X 0,Y 439.691,Z 224.714,A -85,B 0,C 180,E1 -8910,E2 -8910} C_VEL
LIN {X 0,Y 439.61,Z 224.722,A -85,B 0,C 180,E1 -8912.749,E2 -8912.749} C_VEL
LIN {X 0,Y 439.563,Z 224.728,A -85,B 0,C 180,E1 -8916.426,E2 -8916.426} C_VEL
LIN {X 0,Y 439.497,Z 224.738,A -85,B 0,C 180,E1 -8919.201,E2 -8919.201} C_VEL
LIN {X 0,Y 439.468,Z 224.74,A -85,B 0,C 180,E1 -8922.937,E2 -8922.937} C_VEL
LIN {X 0,Y 439.447,Z 224.743,A -85,B 0,C 180,E1 -8926.347,E2 -8926.347} C_VEL
LIN {X 0,Y 439.404,Z 224.754,A -85,B 0,C 180,E1 -8929.626,E2 -8929.626} C_VEL
LIN {X 0,Y 439.365,Z 224.754,A -85,B 0,C 180,E1 -8932.575,E2 -8932.575} C_VEL
LIN {X 0,Y 439.379,Z 224.756,A -85,B 0,C 180,E1 -8935.586,E2 -8935.586} C_VEL
LIN {X 0,Y 439.401,Z 224.75,A -85,B 0,C 180,E1 -8938.674,E2 -8938.674} C_VEL
LIN {X 0,Y 439.371,Z 224.755,A -85,B 0,C 180,E1 -8942.03,E2 -8942.03} C_VEL
LIN {X 0,Y 439.394,Z 224.752,A -85,B 0,C 180,E1 -8945.34,E2 -8945.34} C_VEL
LIN {X 0,Y 439.369,Z 224.754,A -85,B 0,C 180,E1 -8948.596,E2 -8948.596} C_VEL
LIN {X 0,Y 439.381,Z 224.753,A -85,B 0,C 180,E1 -8951.255,E2 -8951.255} C_VEL
LIN {X 0,Y 439.398,Z 224.751,A -85,B 0,C 180,E1 -8954.729,E2 -8954.729} C_VEL
LIN {X 0,Y 439.395,Z 224.753,A -85,B 0,C 180,E1 -8957.795,E2 -8957.795} C_VEL
LIN {X 0,Y 439.409,Z 224.75,A -85,B 0,C 180,E1 -8960.225,E2 -8960.225} C_VEL
LIN {X 0,Y 439.373,Z 224.757,A -85,B 0,C 180,E1 -8963.712,E2 -8963.712} C_VEL
LIN {X 0,Y 439.371,Z 224.754,A -85,B 0,C 180,E1 -8967.054,E2 -8967.054} C_VEL
LIN {X 0,Y 439.38,Z 224.753,A -85,B 0,C 180,E1 -8970.274,E2 -8970.274} C_VEL
LIN {X 0,Y 439.426,Z 224.748,A -85,B 0,C 180,E1 -8973.396,E2 -8973.396} C_VEL
LIN {X 0,Y 439.385,Z 224.753,A -85,B 0,C 180,E1 -8976.429,E2 -8976.429} C_VEL
LIN {X 0,Y 439.386,Z 224.753,A -85,B 0,C 180,E1 -8979.397,E2 -8979.397} C_VEL
LIN {X 0,Y 439.428,Z 224.748,A -85,B 0,C 180,E1 -8982.309,E2 -8982.309} C_VEL
LIN {X 0,Y 439.445,Z 224.745,A -85,B 0,C 180,E1 -8985.174,E2 -8985.174} C_VEL
LIN {X 0,Y 439.481,Z 224.741,A -85,B 0,C 180,E1 -8988.001,E2 -8988.001} C_VEL
LIN {X 0,Y 439.545,Z 224.734,A -85,B 0,C 180,E1 -8991.726,E2 -8991.726} C_VEL
LIN {X 0,Y 439.619,Z 224.725,A -85,B 0,C 180,E1 -8994.496,E2 -8994.496} C_VEL
LIN {X 0,Y 439.633,Z 224.722,A -85,B 0,C 180,E1 -8998.168,E2 -8998.168} C_VEL
LIN {X 0,Y 439.759,Z 224.706,A -85,B 0,C 180,E1 -9000,E2 -9000} C_VEL
LIN {X 0,Y 439.653,Z 224.721,A -85,B 0,C 180,E1 -9002.749,E2 -9002.749} C_VEL
LIN {X 0,Y 439.616,Z 224.726,A -85,B 0,C 180,E1 -9006.425,E2 -9006.425} C_VEL
LIN {X 0,Y 439.497,Z 224.738,A -85,B 0,C 180,E1 -9009.202,E2 -9009.202} C_VEL
LIN {X 0,Y 439.463,Z 224.743,A -85,B 0,C 180,E1 -9012.938,E2 -9012.938} C_VEL
LIN {X 0,Y 439.445,Z 224.747,A -85,B 0,C 180,E1 -9016.349,E2 -9016.349} C_VEL
LIN {X 0,Y 439.4,Z 224.751,A -85,B 0,C 180,E1 -9019.626,E2 -9019.626} C_VEL
LIN {X 0,Y 439.363,Z 224.759,A -85,B 0,C 180,E1 -9022.576,E2 -9022.576} C_VEL
LIN {X 0,Y 439.403,Z 224.75,A -85,B 0,C 180,E1 -9025.585,E2 -9025.585} C_VEL
LIN {X 0,Y 439.415,Z 224.751,A -85,B 0,C 180,E1 -9028.674,E2 -9028.674} C_VEL
LIN {X 0,Y 439.368,Z 224.754,A -85,B 0,C 180,E1 -9032.031,E2 -9032.031} C_VEL
LIN {X 0,Y 439.394,Z 224.75,A -85,B 0,C 180,E1 -9035.341,E2 -9035.341} C_VEL
LIN {X 0,Y 439.377,Z 224.757,A -85,B 0,C 180,E1 -9038.596,E2 -9038.596} C_VEL
LIN {X 0,Y 439.387,Z 224.751,A -85,B 0,C 180,E1 -9041.257,E2 -9041.257} C_VEL
LIN {X 0,Y 439.4,Z 224.752,A -85,B 0,C 180,E1 -9044.73,E2 -9044.73} C_VEL
LIN {X 0,Y 439.395,Z 224.749,A -85,B 0,C 180,E1 -9047.796,E2 -9047.796} C_VEL
LIN {X 0,Y 439.429,Z 224.748,A -85,B 0,C 180,E1 -9050.228,E2 -9050.228} C_VEL
LIN {X 0,Y 439.371,Z 224.752,A -85,B 0,C 180,E1 -9053.713,E2 -9053.713} C_VEL
LIN {X 0,Y 439.373,Z 224.757,A -85,B 0,C 180,E1 -9057.054,E2 -9057.054} C_VEL
LIN {X 0,Y 439.382,Z 224.755,A -85,B 0,C 180,E1 -9060.275,E2 -9060.275} C_VEL
LIN {X 0,Y 439.442,Z 224.837,A -85,B 0,C 180,E1 -9063.487,E2 -9063.487} C_VEL
LIN {X 0,Y 441.848,Z 237.186,A -85,B 0,C 180,E1 -9066.072,E2 -9066.072} C_VEL
LIN {X 0,Y 441.845,Z 242.063,A -85,B 0,C 180,E1 -9067.025,E2 -9067.025} C_VEL
LIN {X 0,Y 440.962,Z 258.224,A -85,B 0,C 180,E1 -9070.109,E2 -9070.109} C_VEL
LIN {X 0,Y 440.46,Z 267.736,A -85,B 0,C 180,E1 -9071.904,E2 -9071.904} C_VEL
LIN {X 0,Y 443.972,Z 290.276,A -85,B 0,C 180,E1 -9072.437,E2 -9072.437} C_VEL
LIN {X 0,Y 443.095,Z 375.592,A -85,B 0,C 180,E1 -9073.855,E2 -9073.855} C_VEL
LIN {X 0,Y 442.678,Z 388.944,A -85,B 0,C 180,E1 -9074.254,E2 -9074.254} C_VEL
LIN {X 0,Y 442.175,Z 401.161,A -85,B 0,C 180,E1 -9074.796,E2 -9074.796} C_VEL
LIN {X 0,Y 441.574,Z 412.666,A -85,B 0,C 180,E1 -9075.483,E2 -9075.483} C_VEL
LIN {X 0,Y 441.004,Z 423.765,A -85,B 0,C 180,E1 -9076.341,E2 -9076.341} C_VEL
LIN {X 0,Y 440.335,Z 435.054,A -85,B 0,C 180,E1 -9077.44,E2 -9077.44} C_VEL
LIN {X 0,Y 439.849,Z 443.704,A -85,B 0,C 180,E1 -9078.479,E2 -9078.479} C_VEL
LIN {X 0,Y 439.309,Z 451.672,A -85,B 0,C 180,E1 -9079.632,E2 -9079.632} C_VEL
LIN {X 0,Y 438.892,Z 459.467,A -85,B 0,C 180,E1 -9081.018,E2 -9081.018} C_VEL
LIN {X 0,Y 438.552,Z 466.62,A -85,B 0,C 180,E1 -9082.634,E2 -9082.634} C_VEL
LIN {X 0,Y 438.381,Z 471.269,A -85,B 0,C 180,E1 -9083.981,E2 -9083.981} C_VEL
LIN {X 0,Y 438.34,Z 475.031,A -85,B 0,C 180,E1 -9085.402,E2 -9085.402} C_VEL
LIN {X 0,Y 438.279,Z 476.911,A -85,B 0,C 180,E1 -9086.323,E2 -9086.323} C_VEL
LIN {X 0,Y 438.34,Z 478.327,A -85,B 0,C 180,E1 -9087.243,E2 -9087.243} C_VEL
LIN {X 0,Y 438.252,Z 479.943,A -85,B 0,C 180,E1 -9089.081,E2 -9089.081} C_VEL
LIN {X 0,Y 438.254,Z 480.167,A -85,B 0,C 180,E1 -9090,E2 -9090} C_VEL
LIN {X 0,Y 438.252,Z 479.957,A -85,B 0,C 180,E1 -9090.919,E2 -9090.919} C_VEL
LIN {X 0,Y 438.34,Z 478.353,A -85,B 0,C 180,E1 -9092.757,E2 -9092.757} C_VEL
LIN {X 0,Y 438.279,Z 476.954,A -85,B 0,C 180,E1 -9093.678,E2 -9093.678} C_VEL
LIN {X 0,Y 438.382,Z 474.013,A -85,B 0,C 180,E1 -9095.059,E2 -9095.059} C_VEL
LIN {X 0,Y 438.448,Z 470.031,A -85,B 0,C 180,E1 -9096.443,E2 -9096.443} C_VEL
LIN {X 0,Y 438.684,Z 463.914,A -85,B 0,C 180,E1 -9098.058,E2 -9098.058} C_VEL
LIN {X 0,Y 439.041,Z 457.228,A -85,B 0,C 180,E1 -9099.444,E2 -9099.444} C_VEL
LIN {X 0,Y 439.488,Z 448.935,A -85,B 0,C 180,E1 -9100.83,E2 -9100.83} C_VEL
LIN {X 0,Y 440.075,Z 440.446,A -85,B 0,C 180,E1 -9101.982,E2 -9101.982} C_VEL
LIN {X 0,Y 440.755,Z 430.427,A -85,B 0,C 180,E1 -9103.087,E2 -9103.087} C_VEL
LIN {X 0,Y 441.202,Z 421.018,A -85,B 0,C 180,E1 -9103.941,E2 -9103.941} C_VEL
LIN {X 0,Y 441.823,Z 410.004,A -85,B 0,C 180,E1 -9104.745,E2 -9104.745} C_VEL
LIN {X 0,Y 442.41,Z 397.819,A -85,B 0,C 180,E1 -9105.432,E2 -9105.432} C_VEL
LIN {X 0,Y 442.97,Z 385.12,A -85,B 0,C 180,E1 -9105.943,E2 -9105.943} C_VEL
LIN {X 0,Y 443.371,Z 371.797,A -85,B 0,C 180,E1 -9106.282,E2 -9106.282} C_VEL
LIN {X 0,Y 444.053,Z 289.201,A -85,B 0,C 180,E1 -9107.655,E2 -9107.655} C_VEL
LIN {X 0,Y 440.488,Z 267.221,A -85,B 0,C 180,E1 -9108.205,E2 -9108.205} C_VEL
LIN {X 0,Y 441.327,Z 250.972,A -85,B 0,C 180,E1 -9111.241,E2 -9111.241} C_VEL
LIN {X 0,Y 441.927,Z 238.13,A -85,B 0,C 180,E1 -9113.675,E2 -9113.675} C_VEL
LIN {X 0,Y 439.791,Z 226.617,A -85,B 0,C 180,E1 -9116.046,E2 -9116.046} C_VEL
LIN {X 0,Y 439.404,Z 224.754,A -85,B 0,C 180,E1 -9116.458,E2 -9116.458} C_VEL
LIN {X 0,Y 439.418,Z 224.749,A -85,B 0,C 180,E1 -9118.673,E2 -9118.673} C_VEL
LIN {X 0,Y 439.371,Z 224.757,A -85,B 0,C 180,E1 -9122.03,E2 -9122.03} C_VEL
LIN {X 0,Y 439.394,Z 224.756,A -85,B 0,C 180,E1 -9125.34,E2 -9125.34} C_VEL
LIN {X 0,Y 439.377,Z 224.752,A -85,B 0,C 180,E1 -9128.595,E2 -9128.595} C_VEL
LIN {X 0,Y 439.389,Z 224.756,A -85,B 0,C 180,E1 -9131.257,E2 -9131.257} C_VEL
LIN {X 0,Y 439.405,Z 224.75,A -85,B 0,C 180,E1 -9134.729,E2 -9134.729} C_VEL
LIN {X 0,Y 439.396,Z 224.748,A -85,B 0,C 180,E1 -9137.796,E2 -9137.796} C_VEL
LIN {X 0,Y 439.41,Z 224.747,A -85,B 0,C 180,E1 -9140.225,E2 -9140.225} C_VEL
LIN {X 0,Y 439.375,Z 224.751,A -85,B 0,C 180,E1 -9143.713,E2 -9143.713} C_VEL
LIN {X 0,Y 439.373,Z 224.757,A -85,B 0,C 180,E1 -9147.054,E2 -9147.054} C_VEL
LIN {X 0,Y 439.382,Z 224.75,A -85,B 0,C 180,E1 -9150.274,E2 -9150.274} C_VEL
LIN {X 0,Y 439.428,Z 224.748,A -85,B 0,C 180,E1 -9153.396,E2 -9153.396} C_VEL
LIN {X 0,Y 439.386,Z 224.749,A -85,B 0,C 180,E1 -9156.43,E2 -9156.43} C_VEL
LIN {X 0,Y 439.388,Z 224.752,A -85,B 0,C 180,E1 -9159.397,E2 -9159.397} C_VEL
LIN {X 0,Y 439.43,Z 224.741,A -85,B 0,C 180,E1 -9162.309,E2 -9162.309} C_VEL
LIN {X 0,Y 439.447,Z 224.741,A -85,B 0,C 180,E1 -9165.174,E2 -9165.174} C_VEL
LIN {X 0,Y 439.483,Z 224.737,A -85,B 0,C 180,E1 -9168.001,E2 -9168.001} C_VEL
LIN {X 0,Y 439.547,Z 224.728,A -85,B 0,C 180,E1 -9171.726,E2 -9171.726} C_VEL
LIN {X 0,Y 439.616,Z 224.723,A -85,B 0,C 180,E1 -9174.496,E2 -9174.496} C_VEL
LIN {X 0,Y 439.635,Z 224.719,A -85,B 0,C 180,E1 -9178.168,E2 -9178.168} C_VEL
LIN {X 0,Y 439.761,Z 224.698,A -85,B 0,C 180,E1 -9180,E2 -9180} C_VEL
LIN {X 0,Y 439.653,Z 224.721,A -85,B 0,C 180,E1 -9182.749,E2 -9182.749} C_VEL
LIN {X 0,Y 439.612,Z 224.725,A -85,B 0,C 180,E1 -9186.425,E2 -9186.425} C_VEL
LIN {X 0,Y 439.499,Z 224.738,A -85,B 0,C 180,E1 -9189.202,E2 -9189.202} C_VEL
LIN {X 0,Y 439.465,Z 224.745,A -85,B 0,C 180,E1 -9192.938,E2 -9192.938} C_VEL
LIN {X 0,Y 439.447,Z 224.744,A -85,B 0,C 180,E1 -9196.349,E2 -9196.349} C_VEL
LIN {X 0,Y 439.402,Z 224.748,A -85,B 0,C 180,E1 -9199.626,E2 -9199.626} C_VEL
LIN {X 0,Y 439.364,Z 224.76,A -85,B 0,C 180,E1 -9202.576,E2 -9202.576} C_VEL
LIN {X 0,Y 439.38,Z 224.751,A -85,B 0,C 180,E1 -9205.587,E2 -9205.587} C_VEL
LIN {X 0,Y 439.399,Z 224.748,A -85,B 0,C 180,E1 -9208.675,E2 -9208.675} C_VEL
LIN {X 0,Y 439.368,Z 224.754,A -85,B 0,C 180,E1 -9212.03,E2 -9212.03} C_VEL
LIN {X 0,Y 439.389,Z 224.753,A -85,B 0,C 180,E1 -9215.34,E2 -9215.34} C_VEL
LIN {X 0,Y 439.357,Z 224.76,A -85,B 0,C 180,E1 -9218.598,E2 -9218.598} C_VEL
LIN {X 0,Y 439.373,Z 224.757,A -85,B 0,C 180,E1 -9222.207,E2 -9222.207} C_VEL
LIN {X 0,Y 439.418,Z 224.922,A -85,B 0,C 180,E1 -9222.689,E2 -9222.689} C_VEL
LIN {X 0,Y 441.036,Z 233.326,A -85,B 0,C 180,E1 -9224.52,E2 -9224.52} C_VEL
LIN {X 0,Y 440.827,Z 242.631,A -85,B 0,C 180,E1 -9226.408,E2 -9226.408} C_VEL
LIN {X 0,Y 440.71,Z 244.964,A -85,B 0,C 180,E1 -9226.879,E2 -9226.879} C_VEL
LIN {X 0,Y 444.394,Z 263.32,A -85,B 0,C 180,E1 -9227.357,E2 -9227.357} C_VEL
LIN {X 0,Y 443.29,Z 353.003,A -85,B 0,C 180,E1 -9228.857,E2 -9228.857} C_VEL
LIN {X 0,Y 442.973,Z 366.317,A -85,B 0,C 180,E1 -9229.272,E2 -9229.272} C_VEL
LIN {X 0,Y 442.527,Z 378.906,A -85,B 0,C 180,E1 -9229.853,E2 -9229.853} C_VEL
LIN {X 0,Y 441.962,Z 390.973,A -85,B 0,C 180,E1 -9230.614,E2 -9230.614} C_VEL
LIN {X 0,Y 441.357,Z 401.666,A -85,B 0,C 180,E1 -9231.476,E2 -9231.476} C_VEL
LIN {X 0,Y 440.692,Z 412.399,A -85,B 0,C 180,E1 -9232.555,E2 -9232.555} C_VEL
LIN {X 0,Y 440.083,Z 422.108,A -85,B 0,C 180,E1 -9233.781,E2 -9233.781} C_VEL
LIN {X 0,Y 439.541,Z 430.78,A -85,B 0,C 180,E1 -9235.137,E2 -9235.137} C_VEL
LIN {X 0,Y 439.15,Z 436.973,A -85,B 0,C 180,E1 -9236.325,E2 -9236.325} C_VEL
LIN {X 0,Y 438.854,Z 442.255,A -85,B 0,C 180,E1 -9237.556,E2 -9237.556} C_VEL
LIN {X 0,Y 438.6,Z 447.674,A -85,B 0,C 180,E1 -9239.152,E2 -9239.152} C_VEL
LIN {X 0,Y 438.398,Z 451.574,A -85,B 0,C 180,E1 -9240.729,E2 -9240.729} C_VEL
LIN {X 0,Y 438.205,Z 454.156,A -85,B 0,C 180,E1 -9242.283,E2 -9242.283} C_VEL
LIN {X 0,Y 438.137,Z 455.621,A -85,B 0,C 180,E1 -9243.933,E2 -9243.933} C_VEL
LIN {X 0,Y 438.098,Z 455.694,A -85,B 0,C 180,E1 -9245.843,E2 -9245.843} C_VEL
LIN {X 0,Y 438.157,Z 454.604,A -85,B 0,C 180,E1 -9247.359,E2 -9247.359} C_VEL
LIN {X 0,Y 438.275,Z 453.102,A -85,B 0,C 180,E1 -9248.446,E2 -9248.446} C_VEL
LIN {X 0,Y 438.431,Z 450.466,A -85,B 0,C 180,E1 -9249.778,E2 -9249.778} C_VEL
LIN {X 0,Y 437.858,Z 448.698,A -85,B 0,C 180,E1 -9250.511,E2 -9250.511} C_VEL
LIN {X 0,Y 435.15,Z 445.362,A -85,B 0,C 180,E1 -9251.684,E2 -9251.684} C_VEL
LIN {X 0,Y 432.472,Z 441.356,A -85,B 0,C 180,E1 -9252.834,E2 -9252.834} C_VEL
LIN {X 0,Y 431.96,Z 438.51,A -85,B 0,C 180,E1 -9253.52,E2 -9253.52} C_VEL
LIN {X 0,Y 432.411,Z 431.523,A -85,B 0,C 180,E1 -9254.927,E2 -9254.927} C_VEL
LIN {X 0,Y 432.911,Z 423.887,A -85,B 0,C 180,E1 -9256.169,E2 -9256.169} C_VEL
LIN {X 0,Y 433.553,Z 413.975,A -85,B 0,C 180,E1 -9257.478,E2 -9257.478} C_VEL
LIN {X 0,Y 434.187,Z 403.787,A -85,B 0,C 180,E1 -9258.563,E2 -9258.563} C_VEL
LIN {X 0,Y 434.86,Z 392.384,A -85,B 0,C 180,E1 -9259.524,E2 -9259.524} C_VEL
LIN {X 0,Y 435.435,Z 380.345,A -85,B 0,C 180,E1 -9260.317,E2 -9260.317} C_VEL
LIN {X 0,Y 435.843,Z 368.703,A -85,B 0,C 180,E1 -9260.896,E2 -9260.896} C_VEL
LIN {X 0,Y 436.247,Z 355.582,A -85,B 0,C 180,E1 -9261.342,E2 -9261.342} C_VEL
LIN {X 0,Y 436.552,Z 337.077,A -85,B 0,C 180,E1 -9261.698,E2 -9261.698} C_VEL
LIN {X 0,Y 437.289,Z 263.343,A -85,B 0,C 180,E1 -9262.932,E2 -9262.932} C_VEL
LIN {X 0,Y 433.759,Z 245.178,A -85,B 0,C 180,E1 -9263.4,E2 -9263.4} C_VEL
LIN {X 0,Y 434.054,Z 235.177,A -85,B 0,C 180,E1 -9265.589,E2 -9265.589} C_VEL
LIN {X 0,Y 432.578,Z 225.604,A -85,B 0,C 180,E1 -9267.847,E2 -9267.847} C_VEL
LIN {X 0,Y 432.642,Z 225.592,A -85,B 0,C 180,E1 -9270,E2 -9270} C_VEL
LIN {X 0,Y 432.563,Z 225.601,A -85,B 0,C 180,E1 -9272.794,E2 -9272.794} C_VEL
LIN {X 0,Y 432.575,Z 225.604,A -85,B 0,C 180,E1 -9275.594,E2 -9275.594} C_VEL
LIN {X 0,Y 432.466,Z 225.612,A -85,B 0,C 180,E1 -9278.41,E2 -9278.41} C_VEL
LIN {X 0,Y 432.462,Z 225.614,A -85,B 0,C 180,E1 -9282.196,E2 -9282.196} C_VEL
LIN {X 0,Y 432.428,Z 225.62,A -85,B 0,C 180,E1 -9286.039,E2 -9286.039} C_VEL
LIN {X 0,Y 432.388,Z 225.626,A -85,B 0,C 180,E1 -9289.484,E2 -9289.484} C_VEL
LIN {X 0,Y 432.318,Z 225.631,A -85,B 0,C 180,E1 -9292.964,E2 -9292.964} C_VEL
LIN {X 0,Y 432.339,Z 225.629,A -85,B 0,C 180,E1 -9295.002,E2 -9295.002} C_VEL
LIN {X 0,Y 432.348,Z 225.629,A -85,B 0,C 180,E1 -9298.125,E2 -9298.125} C_VEL
LIN {X 0,Y 432.322,Z 225.633,A -85,B 0,C 180,E1 -9301.346,E2 -9301.346} C_VEL
LIN {X 0,Y 432.34,Z 225.63,A -85,B 0,C 180,E1 -9304.677,E2 -9304.677} C_VEL
LIN {X 0,Y 432.332,Z 225.631,A -85,B 0,C 180,E1 -9308.15,E2 -9308.15} C_VEL
LIN {X 0,Y 432.324,Z 225.635,A -85,B 0,C 180,E1 -9311.6,E2 -9311.6} C_VEL
LIN {X 0,Y 432.333,Z 225.631,A -85,B 0,C 180,E1 -9314.347,E2 -9314.347} C_VEL
LIN {X 0,Y 432.319,Z 225.632,A -85,B 0,C 180,E1 -9317.015,E2 -9317.015} C_VEL
LIN {X 0,Y 432.332,Z 225.633,A -85,B 0,C 180,E1 -9319.82,E2 -9319.82} C_VEL
LIN {X 0,Y 432.306,Z 225.634,A -85,B 0,C 180,E1 -9323.022,E2 -9323.022} C_VEL
LIN {X 0,Y 432.358,Z 225.629,A -85,B 0,C 180,E1 -9325.996,E2 -9325.996} C_VEL
LIN {X 0,Y 432.346,Z 225.631,A -85,B 0,C 180,E1 -9329.489,E2 -9329.489} C_VEL
LIN {X 0,Y 432.389,Z 225.624,A -85,B 0,C 180,E1 -9332.928,E2 -9332.928} C_VEL
LIN {X 0,Y 432.37,Z 225.627,A -85,B 0,C 180,E1 -9336.023,E2 -9336.023} C_VEL
LIN {X 0,Y 432.348,Z 225.629,A -85,B 0,C 180,E1 -9339.046,E2 -9339.046} C_VEL
LIN {X 0,Y 432.375,Z 225.627,A -85,B 0,C 180,E1 -9342.011,E2 -9342.011} C_VEL
LIN {X 0,Y 432.393,Z 225.624,A -85,B 0,C 180,E1 -9344.926,E2 -9344.926} C_VEL
LIN {X 0,Y 432.457,Z 225.617,A -85,B 0,C 180,E1 -9347.803,E2 -9347.803} C_VEL
LIN {X 0,Y 432.489,Z 225.613,A -85,B 0,C 180,E1 -9351.59,E2 -9351.59} C_VEL
LIN {X 0,Y 432.596,Z 225.6,A -85,B 0,C 180,E1 -9354.406,E2 -9354.406} C_VEL
LIN {X 0,Y 432.603,Z 225.598,A -85,B 0,C 180,E1 -9358.138,E2 -9358.138} C_VEL
LIN {X 0,Y 432.729,Z 225.582,A -85,B 0,C 180,E1 -9360,E2 -9360} C_VEL
LIN {X 0,Y 432.602,Z 225.598,A -85,B 0,C 180,E1 -9362.794,E2 -9362.794} C_VEL
LIN {X 0,Y 432.571,Z 225.604,A -85,B 0,C 180,E1 -9366.53,E2 -9366.53} C_VEL
LIN {X 0,Y 432.44,Z 225.617,A -85,B 0,C 180,E1 -9369.353,E2 -9369.353} C_VEL
LIN {X 0,Y 432.428,Z 225.62,A -85,B 0,C 180,E1 -9372.804,E2 -9372.804} C_VEL
LIN {X 0,Y 432.41,Z 225.624,A -85,B 0,C 180,E1 -9376.479,E2 -9376.479} C_VEL
LIN {X 0,Y 432.336,Z 225.63,A -85,B 0,C 180,E1 -9379.961,E2 -9379.961} C_VEL
LIN {X 0,Y 432.317,Z 225.633,A -85,B 0,C 180,E1 -9382.964,E2 -9382.964} C_VEL
LIN {X 0,Y 432.362,Z 225.627,A -85,B 0,C 180,E1 -9386.033,E2 -9386.033} C_VEL
LIN {X 0,Y 432.34,Z 225.629,A -85,B 0,C 180,E1 -9389.188,E2 -9389.188} C_VEL
LIN {X 0,Y 432.321,Z 225.635,A -85,B 0,C 180,E1 -9392.443,E2 -9392.443} C_VEL
LIN {X 0,Y 432.343,Z 225.629,A -85,B 0,C 180,E1 -9395.632,E2 -9395.632} C_VEL
LIN {X 0,Y 432.345,Z 225.628,A -85,B 0,C 180,E1 -9399.343,E2 -9399.343} C_VEL
LIN {X 0,Y 432.332,Z 225.63,A -85,B 0,C 180,E1 -9401.797,E2 -9401.797} C_VEL
LIN {X 0,Y 432.332,Z 225.633,A -85,B 0,C 180,E1 -9404.348,E2 -9404.348} C_VEL
LIN {X 0,Y 432.319,Z 225.632,A -85,B 0,C 180,E1 -9407.016,E2 -9407.016} C_VEL
LIN {X 0,Y 432.335,Z 225.629,A -85,B 0,C 180,E1 -9409.821,E2 -9409.821} C_VEL
LIN {X 0,Y 432.304,Z 225.633,A -85,B 0,C 180,E1 -9413.022,E2 -9413.022} C_VEL
LIN {X 0,Y 432.359,Z 225.626,A -85,B 0,C 180,E1 -9415.997,E2 -9415.997} C_VEL
LIN {X 0,Y 432.348,Z 225.629,A -85,B 0,C 180,E1 -9419.49,E2 -9419.49} C_VEL
LIN {X 0,Y 432.391,Z 225.629,A -85,B 0,C 180,E1 -9422.929,E2 -9422.929} C_VEL
LIN {X 0,Y 432.407,Z 225.794,A -85,B 0,C 180,E1 -9423.269,E2 -9423.269} C_VEL
LIN {X 0,Y 435.023,Z 239.49,A -85,B 0,C 180,E1 -9426.179,E2 -9426.179} C_VEL
LIN {X 0,Y 434.292,Z 253.42,A -85,B 0,C 180,E1 -9428.896,E2 -9428.896} C_VEL
LIN {X 0,Y 433.5,Z 267.584,A -85,B 0,C 180,E1 -9431.62,E2 -9431.62} C_VEL
LIN {X 0,Y 437.17,Z 291.101,A -85,B 0,C 180,E1 -9432.182,E2 -9432.182} C_VEL
LIN {X 0,Y 436.235,Z 376.144,A -85,B 0,C 180,E1 -9433.625,E2 -9433.625} C_VEL
LIN {X 0,Y 435.769,Z 390.002,A -85,B 0,C 180,E1 -9434.058,E2 -9434.058} C_VEL
LIN {X 0,Y 435.269,Z 401.896,A -85,B 0,C 180,E1 -9434.609,E2 -9434.609} C_VEL
LIN {X 0,Y 434.58,Z 413.945,A -85,B 0,C 180,E1 -9435.364,E2 -9435.364} C_VEL
LIN {X 0,Y 433.972,Z 425.232,A -85,B 0,C 180,E1 -9436.279,E2 -9436.279} C_VEL
LIN {X 0,Y 433.313,Z 435.839,A -85,B 0,C 180,E1 -9437.352,E2 -9437.352} C_VEL
LIN {X 0,Y 432.738,Z 445.158,A -85,B 0,C 180,E1 -9438.525,E2 -9438.525} C_VEL
LIN {X 0,Y 432.188,Z 452.829,A -85,B 0,C 180,E1 -9439.696,E2 -9439.696} C_VEL
LIN {X 0,Y 431.806,Z 460.349,A -85,B 0,C 180,E1 -9441.105,E2 -9441.105} C_VEL
LIN {X 0,Y 431.498,Z 466.388,A -85,B 0,C 180,E1 -9442.513,E2 -9442.513} C_VEL
LIN {X 0,Y 431.281,Z 471.478,A -85,B 0,C 180,E1 -9444.023,E2 -9444.023} C_VEL
LIN {X 0,Y 431.269,Z 474.815,A -85,B 0,C 180,E1 -9445.327,E2 -9445.327} C_VEL
LIN {X 0,Y 431.186,Z 476.699,A -85,B 0,C 180,E1 -9446.262,E2 -9446.262} C_VEL
LIN {X 0,Y 431.236,Z 478.12,A -85,B 0,C 180,E1 -9447.198,E2 -9447.198} C_VEL
LIN {X 0,Y 431.203,Z 479.127,A -85,B 0,C 180,E1 -9448.132,E2 -9448.132} C_VEL
LIN {X 0,Y 431.168,Z 479.97,A -85,B 0,C 180,E1 -9450,E2 -9450} C_VEL
LIN {X 0,Y 431.169,Z 479.764,A -85,B 0,C 180,E1 -9450.934,E2 -9450.934} C_VEL
LIN {X 0,Y 431.203,Z 479.159,A -85,B 0,C 180,E1 -9451.868,E2 -9451.868} C_VEL
LIN {X 0,Y 431.235,Z 478.164,A -85,B 0,C 180,E1 -9452.803,E2 -9452.803} C_VEL
LIN {X 0,Y 431.186,Z 476.768,A -85,B 0,C 180,E1 -9453.738,E2 -9453.738} C_VEL
LIN {X 0,Y 431.293,Z 473.83,A -85,B 0,C 180,E1 -9455.142,E2 -9455.142} C_VEL
LIN {X 0,Y 431.376,Z 469.853,A -85,B 0,C 180,E1 -9456.549,E2 -9456.549} C_VEL
LIN {X 0,Y 431.625,Z 463.743,A -85,B 0,C 180,E1 -9458.191,E2 -9458.191} C_VEL
LIN {X 0,Y 431.989,Z 457.061,A -85,B 0,C 180,E1 -9459.599,E2 -9459.599} C_VEL
LIN {X 0,Y 432.471,Z 448.773,A -85,B 0,C 180,E1 -9461.008,E2 -9461.008} C_VEL
LIN {X 0,Y 433.117,Z 440.292,A -85,B 0,C 180,E1 -9462.178,E2 -9462.178} C_VEL
LIN {X 0,Y 433.786,Z 430.704,A -85,B 0,C 180,E1 -9463.259,E2 -9463.259} C_VEL
LIN {X 0,Y 434.302,Z 420.888,A -85,B 0,C 180,E1 -9464.168,E2 -9464.168} C_VEL
LIN {X 0,Y 434.933,Z 409.891,A -85,B 0,C 180,E1 -9464.984,E2 -9464.984} C_VEL
LIN {X 0,Y 435.577,Z 397.731,A -85,B 0,C 180,E1 -9465.68,E2 -9465.68} C_VEL
LIN {X 0,Y 436.144,Z 385.116,A -85,B 0,C 180,E1 -9466.199,E2 -9466.199} C_VEL
LIN {X 0,Y 436.582,Z 371.941,A -85,B 0,C 180,E1 -9466.543,E2 -9466.543} C_VEL
LIN {X 0,Y 437.316,Z 290.024,A -85,B 0,C 180,E1 -9467.929,E2 -9467.929} C_VEL
LIN {X 0,Y 433.564,Z 267.083,A -85,B 0,C 180,E1 -9468.504,E2 -9468.504} C_VEL
LIN {X 0,Y 434.591,Z 248.253,A -85,B 0,C 180,E1 -9472.085,E2 -9472.085} C_VEL
LIN {X 0,Y 434.968,Z 239.262,A -85,B 0,C 180,E1 -9473.825,E2 -9473.825} C_VEL
LIN {X 0,Y 432.742,Z 227.43,A -85,B 0,C 180,E1 -9476.311,E2 -9476.311} C_VEL
LIN {X 0,Y 432.378,Z 225.63,A -85,B 0,C 180,E1 -9476.731,E2 -9476.731} C_VEL
LIN {X 0,Y 432.344,Z 225.63,A -85,B 0,C 180,E1 -9479.187,E2 -9479.187} C_VEL
LIN {X 0,Y 432.324,Z 225.634,A -85,B 0,C 180,E1 -9482.443,E2 -9482.443} C_VEL
LIN {X 0,Y 432.344,Z 225.631,A -85,B 0,C 180,E1 -9485.631,E2 -9485.631} C_VEL
LIN {X 0,Y 432.34,Z 225.629,A -85,B 0,C 180,E1 -9488.714,E2 -9488.714} C_VEL
LIN {X 0,Y 432.334,Z 225.629,A -85,B 0,C 180,E1 -9491.797,E2 -9491.797} C_VEL
LIN {X 0,Y 432.34,Z 225.629,A -85,B 0,C 180,E1 -9494.346,E2 -9494.346} C_VEL
LIN {X 0,Y 432.32,Z 225.636,A -85,B 0,C 180,E1 -9497.015,E2 -9497.015} C_VEL
LIN {X 0,Y 432.333,Z 225.63,A -85,B 0,C 180,E1 -9499.821,E2 -9499.821} C_VEL
LIN {X 0,Y 432.307,Z 225.636,A -85,B 0,C 180,E1 -9503.022,E2 -9503.022} C_VEL
LIN {X 0,Y 432.359,Z 225.625,A -85,B 0,C 180,E1 -9505.996,E2 -9505.996} C_VEL
LIN {X 0,Y 432.347,Z 225.629,A -85,B 0,C 180,E1 -9509.489,E2 -9509.489} C_VEL
LIN {X 0,Y 432.391,Z 225.621,A -85,B 0,C 180,E1 -9512.928,E2 -9512.928} C_VEL
LIN {X 0,Y 432.371,Z 225.622,A -85,B 0,C 180,E1 -9516.023,E2 -9516.023} C_VEL
LIN {X 0,Y 432.35,Z 225.633,A -85,B 0,C 180,E1 -9519.046,E2 -9519.046} C_VEL
LIN {X 0,Y 432.376,Z 225.619,A -85,B 0,C 180,E1 -9522.011,E2 -9522.011} C_VEL
LIN {X 0,Y 432.395,Z 225.622,A -85,B 0,C 180,E1 -9524.926,E2 -9524.926} C_VEL
LIN {X 0,Y 432.458,Z 225.612,A -85,B 0,C 180,E1 -9527.803,E2 -9527.803} C_VEL
LIN {X 0,Y 432.491,Z 225.608,A -85,B 0,C 180,E1 -9531.59,E2 -9531.59} C_VEL
LIN {X 0,Y 432.593,Z 225.597,A -85,B 0,C 180,E1 -9534.406,E2 -9534.406} C_VEL
LIN {X 0,Y 432.605,Z 225.595,A -85,B 0,C 180,E1 -9538.138,E2 -9538.138} C_VEL
LIN {X 0,Y 432.731,Z 225.573,A -85,B 0,C 180,E1 -9540,E2 -9540} C_VEL
LIN {X 0,Y 432.603,Z 225.598,A -85,B 0,C 180,E1 -9542.794,E2 -9542.794} C_VEL
LIN {X 0,Y 432.568,Z 225.604,A -85,B 0,C 180,E1 -9546.53,E2 -9546.53} C_VEL
LIN {X 0,Y 432.442,Z 225.616,A -85,B 0,C 180,E1 -9549.353,E2 -9549.353} C_VEL
LIN {X 0,Y 432.43,Z 225.621,A -85,B 0,C 180,E1 -9552.804,E2 -9552.804} C_VEL
LIN {X 0,Y 432.412,Z 225.622,A -85,B 0,C 180,E1 -9556.479,E2 -9556.479} C_VEL
LIN {X 0,Y 432.338,Z 225.629,A -85,B 0,C 180,E1 -9559.961,E2 -9559.961} C_VEL
LIN {X 0,Y 432.317,Z 225.633,A -85,B 0,C 180,E1 -9562.965,E2 -9562.965} C_VEL
LIN {X 0,Y 432.339,Z 225.631,A -85,B 0,C 180,E1 -9565.002,E2 -9565.002} C_VEL
LIN {X 0,Y 432.347,Z 225.63,A -85,B 0,C 180,E1 -9568.126,E2 -9568.126} C_VEL
LIN {X 0,Y 432.32,Z 225.631,A -85,B 0,C 180,E1 -9571.346,E2 -9571.346} C_VEL
LIN {X 0,Y 432.336,Z 225.633,A -85,B 0,C 180,E1 -9574.678,E2 -9574.678} C_VEL
LIN {X 0,Y 432.324,Z 225.636,A -85,B 0,C 180,E1 -9578.152,E2 -9578.152} C_VEL
LIN {X 0,Y 432.315,Z 225.635,A -85,B 0,C 180,E1 -9581.8,E2 -9581.8} C_VEL
LIN {X 0,Y 432.368,Z 225.683,A -85,B 0,C 180,E1 -9582.421,E2 -9582.421} C_VEL
LIN {X 0,Y 434.17,Z 235.484,A -85,B 0,C 180,E1 -9584.583,E2 -9584.583} C_VEL
LIN {X 0,Y 433.802,Z 245.237,A -85,B 0,C 180,E1 -9586.568,E2 -9586.568} C_VEL
LIN {X 0,Y 437.611,Z 263.769,A -85,B 0,C 180,E1 -9587.066,E2 -9587.066} C_VEL
LIN {X 0,Y 436.533,Z 352.749,A -85,B 0,C 180,E1 -9588.579,E2 -9588.579} C_VEL
LIN {X 0,Y 436.182,Z 366.287,A -85,B 0,C 180,E1 -9589.003,E2 -9589.003} C_VEL
LIN {X 0,Y 435.748,Z 377.301,A -85,B 0,C 180,E1 -9589.507,E2 -9589.507} C_VEL
LIN {X 0,Y 435.192,Z 388.979,A -85,B 0,C 180,E1 -9590.215,E2 -9590.215} C_VEL
LIN {X 0,Y 434.567,Z 400.06,A -85,B 0,C 180,E1 -9591.086,E2 -9591.086} C_VEL
LIN {X 0,Y 433.875,Z 411.089,A -85,B 0,C 180,E1 -9592.18,E2 -9592.18} C_VEL
LIN {X 0,Y 433.225,Z 421.001,A -85,B 0,C 180,E1 -9593.404,E2 -9593.404} C_VEL
LIN {X 0,Y 432.622,Z 429.903,A -85,B 0,C 180,E1 -9594.781,E2 -9594.781} C_VEL
LIN {X 0,Y 432.149,Z 436.528,A -85,B 0,C 180,E1 -9596.038,E2 -9596.038} C_VEL
LIN {X 0,Y 431.781,Z 442.785,A -85,B 0,C 180,E1 -9597.511,E2 -9597.511} C_VEL
LIN {X 0,Y 431.531,Z 448.123,A -85,B 0,C 180,E1 -9599.135,E2 -9599.135} C_VEL
LIN {X 0,Y 431.322,Z 451.936,A -85,B 0,C 180,E1 -9600.737,E2 -9600.737} C_VEL
LIN {X 0,Y 431.178,Z 453.753,A -85,B 0,C 180,E1 -9601.791,E2 -9601.791} C_VEL
LIN {X 0,Y 431.061,Z 455.051,A -85,B 0,C 180,E1 -9602.838,E2 -9602.838} C_VEL
LIN {X 0,Y 431.057,Z 455.805,A -85,B 0,C 180,E1 -9603.883,E2 -9603.883} C_VEL
LIN {X 0,Y 431.016,Z 456.103,A -85,B 0,C 180,E1 -9604.916,E2 -9604.916} C_VEL
LIN {X 0,Y 431.008,Z 455.892,A -85,B 0,C 180,E1 -9605.943,E2 -9605.943} C_VEL
LIN {X 0,Y 431.035,Z 455.209,A -85,B 0,C 180,E1 -9606.963,E2 -9606.963} C_VEL
LIN {X 0,Y 431.171,Z 453.606,A -85,B 0,C 180,E1 -9608.294,E2 -9608.294} C_VEL
LIN {X 0,Y 431.394,Z 450.328,A -85,B 0,C 180,E1 -9609.994,E2 -9609.994} C_VEL
LIN {X 0,Y 431.581,Z 446.228,A -85,B 0,C 180,E1 -9611.486,E2 -9611.486} C_VEL
LIN {X 0,Y 431.827,Z 440.902,A -85,B 0,C 180,E1 -9612.965,E2 -9612.965} C_VEL
LIN {X 0,Y 431.96,Z 438.51,A -85,B 0,C 180,E1 -9613.52,E2 -9613.52} C_VEL
LIN {X 0,Y 431.488,Z 435.484,A -85,B 0,C 180,E1 -9614.192,E2 -9614.192} C_VEL
LIN {X 0,Y 429.013,Z 430.256,A -85,B 0,C 180,E1 -9615.267,E2 -9615.267} C_VEL
LIN {X 0,Y 426.575,Z 424.408,A -85,B 0,C 180,E1 -9616.29,E2 -9616.29} C_VEL
LIN {X 0,Y 426.159,Z 420.408,A -85,B 0,C 180,E1 -9616.873,E2 -9616.873} C_VEL
LIN {X 0,Y 426.857,Z 410.254,A -85,B 0,C 180,E1 -9618.123,E2 -9618.123} C_VEL
LIN {X 0,Y 427.556,Z 399.111,A -85,B 0,C 180,E1 -9619.223,E2 -9619.223} C_VEL
LIN {X 0,Y 428.337,Z 386.996,A -85,B 0,C 180,E1 -9620.149,E2 -9620.149} C_VEL
LIN {X 0,Y 428.833,Z 374.837,A -85,B 0,C 180,E1 -9620.865,E2 -9620.865} C_VEL
LIN {X 0,Y 429.247,Z 362.862,A -85,B 0,C 180,E1 -9621.378,E2 -9621.378} C_VEL
LIN {X 0,Y 429.554,Z 349.776,A -85,B 0,C 180,E1 -9621.74,E2 -9621.74} C_VEL
LIN {X 0,Y 430.488,Z 264.171,A -85,B 0,C 180,E1 -9623.202,E2 -9623.202} C_VEL
LIN {X 0,Y 426.798,Z 245.316,A -85,B 0,C 180,E1 -9623.707,E2 -9623.707} C_VEL
LIN {X 0,Y 427.149,Z 237.143,A -85,B 0,C 180,E1 -9625.517,E2 -9625.517} C_VEL
LIN {X 0,Y 425.546,Z 226.479,A -85,B 0,C 180,E1 -9628.048,E2 -9628.048} C_VEL
LIN {X 0,Y 425.593,Z 226.469,A -85,B 0,C 180,E1 -9630,E2 -9630} C_VEL
LIN {X 0,Y 425.519,Z 226.48,A -85,B 0,C 180,E1 -9632.84,E2 -9632.84} C_VEL
LIN {X 0,Y 425.53,Z 226.482,A -85,B 0,C 180,E1 -9635.687,E2 -9635.687} C_VEL
LIN {X 0,Y 425.41,Z 226.491,A -85,B 0,C 180,E1 -9638.55,E2 -9638.55} C_VEL
LIN {X 0,Y 425.415,Z 226.491,A -85,B 0,C 180,E1 -9642.401,E2 -9642.401} C_VEL
LIN {X 0,Y 425.388,Z 226.495,A -85,B 0,C 180,E1 -9646.311,E2 -9646.311} C_VEL
LIN {X 0,Y 425.33,Z 226.506,A -85,B 0,C 180,E1 -9649.635,E2 -9649.635} C_VEL
LIN {X 0,Y 425.305,Z 226.507,A -85,B 0,C 180,E1 -9653.365,E2 -9653.365} C_VEL
LIN {X 0,Y 425.302,Z 226.506,A -85,B 0,C 180,E1 -9656.498,E2 -9656.498} C_VEL
LIN {X 0,Y 425.287,Z 226.512,A -85,B 0,C 180,E1 -9659.719,E2 -9659.719} C_VEL
LIN {X 0,Y 425.283,Z 226.508,A -85,B 0,C 180,E1 -9663.047,E2 -9663.047} C_VEL
LIN {X 0,Y 425.281,Z 226.511,A -85,B 0,C 180,E1 -9665.928,E2 -9665.928} C_VEL
LIN {X 0,Y 425.276,Z 226.509,A -85,B 0,C 180,E1 -9669.039,E2 -9669.039} C_VEL
LIN {X 0,Y 425.282,Z 226.511,A -85,B 0,C 180,E1 -9671.956,E2 -9671.956} C_VEL
LIN {X 0,Y 425.284,Z 226.509,A -85,B 0,C 180,E1 -9675.283,E2 -9675.283} C_VEL
LIN {X 0,Y 425.273,Z 226.511,A -85,B 0,C 180,E1 -9678.621,E2 -9678.621} C_VEL
LIN {X 0,Y 425.301,Z 226.506,A -85,B 0,C 180,E1 -9681.101,E2 -9681.101} C_VEL
LIN {X 0,Y 425.299,Z 226.508,A -85,B 0,C 180,E1 -9684.664,E2 -9684.664} C_VEL
LIN {X 0,Y 425.263,Z 226.513,A -85,B 0,C 180,E1 -9688.073,E2 -9688.073} C_VEL
LIN {X 0,Y 425.329,Z 226.504,A -85,B 0,C 180,E1 -9691.367,E2 -9691.367} C_VEL
LIN {X 0,Y 425.294,Z 226.509,A -85,B 0,C 180,E1 -9694.554,E2 -9694.554} C_VEL
LIN {X 0,Y 425.286,Z 226.511,A -85,B 0,C 180,E1 -9697.661,E2 -9697.661} C_VEL
LIN {X 0,Y 425.36,Z 226.5,A -85,B 0,C 180,E1 -9700.704,E2 -9700.704} C_VEL
LIN {X 0,Y 425.386,Z 226.499,A -85,B 0,C 180,E1 -9703.688,E2 -9703.688} C_VEL
LIN {X 0,Y 425.409,Z 226.495,A -85,B 0,C 180,E1 -9707.598,E2 -9707.598} C_VEL
LIN {X 0,Y 425.44,Z 226.49,A -85,B 0,C 180,E1 -9711.45,E2 -9711.45} C_VEL
LIN {X 0,Y 425.552,Z 226.477,A -85,B 0,C 180,E1 -9714.313,E2 -9714.313} C_VEL
LIN {X 0,Y 425.573,Z 226.474,A -85,B 0,C 180,E1 -9718.107,E2 -9718.107} C_VEL
LIN {X 0,Y 425.699,Z 226.458,A -85,B 0,C 180,E1 -9720,E2 -9720} C_VEL
LIN {X 0,Y 425.554,Z 226.476,A -85,B 0,C 180,E1 -9722.84,E2 -9722.84} C_VEL
LIN {X 0,Y 425.529,Z 226.481,A -85,B 0,C 180,E1 -9726.639,E2 -9726.639} C_VEL
LIN {X 0,Y 425.398,Z 226.495,A -85,B 0,C 180,E1 -9729.509,E2 -9729.509} C_VEL
LIN {X 0,Y 425.39,Z 226.496,A -85,B 0,C 180,E1 -9732.904,E2 -9732.904} C_VEL
LIN {X 0,Y 425.359,Z 226.502,A -85,B 0,C 180,E1 -9736.605,E2 -9736.605} C_VEL
LIN {X 0,Y 425.326,Z 226.504,A -85,B 0,C 180,E1 -9739.636,E2 -9739.636} C_VEL
LIN {X 0,Y 425.305,Z 226.505,A -85,B 0,C 180,E1 -9743.365,E2 -9743.365} C_VEL
LIN {X 0,Y 425.345,Z 226.502,A -85,B 0,C 180,E1 -9746.844,E2 -9746.844} C_VEL
LIN {X 0,Y 425.288,Z 226.508,A -85,B 0,C 180,E1 -9749.72,E2 -9749.72} C_VEL
LIN {X 0,Y 425.28,Z 226.509,A -85,B 0,C 180,E1 -9753.048,E2 -9753.048} C_VEL
LIN {X 0,Y 425.281,Z 226.509,A -85,B 0,C 180,E1 -9755.929,E2 -9755.929} C_VEL
LIN {X 0,Y 425.292,Z 226.507,A -85,B 0,C 180,E1 -9759.043,E2 -9759.043} C_VEL
LIN {X 0,Y 425.273,Z 226.513,A -85,B 0,C 180,E1 -9762.653,E2 -9762.653} C_VEL
LIN {X 0,Y 425.26,Z 226.511,A -85,B 0,C 180,E1 -9766.045,E2 -9766.045} C_VEL
LIN {X 0,Y 425.274,Z 226.513,A -85,B 0,C 180,E1 -9768.622,E2 -9768.622} C_VEL
LIN {X 0,Y 425.309,Z 226.504,A -85,B 0,C 180,E1 -9771.103,E2 -9771.103} C_VEL
LIN {X 0,Y 425.298,Z 226.51,A -85,B 0,C 180,E1 -9774.664,E2 -9774.664} C_VEL
LIN {X 0,Y 425.265,Z 226.511,A -85,B 0,C 180,E1 -9778.074,E2 -9778.074} C_VEL
LIN {X 0,Y 425.331,Z 226.504,A -85,B 0,C 180,E1 -9781.368,E2 -9781.368} C_VEL
LIN {X 0,Y 425.364,Z 226.552,A -85,B 0,C 180,E1 -9783.003,E2 -9783.003} C_VEL
LIN {X 0,Y 428.057,Z 240.505,A -85,B 0,C 180,E1 -9786.024,E2 -9786.024} C_VEL
LIN {X 0,Y 427.664,Z 249.378,A -85,B 0,C 180,E1 -9787.792,E2 -9787.792} C_VEL
LIN {X 0,Y 426.613,Z 265.944,A -85,B 0,C 180,E1 -9791.038,E2 -9791.038} C_VEL
LIN {X 0,Y 426.533,Z 267.405,A -85,B 0,C 180,E1 -9791.323,E2 -9791.323} C_VEL
LIN {X 0,Y 430.38,Z 292.243,A -85,B 0,C 180,E1 -9791.925,E2 -9791.925} C_VEL
LIN {X 0,Y 429.444,Z 375.552,A -85,B 0,C 180,E1 -9793.358,E2 -9793.358} C_VEL
LIN {X 0,Y 428.98,Z 388.777,A -85,B 0,C 180,E1 -9793.768,E2 -9793.768} C_VEL
LIN {X 0,Y 428.392,Z 401.499,A -85,B 0,C 180,E1 -9794.356,E2 -9794.356} C_VEL
LIN {X 0,Y 427.705,Z 413.611,A -85,B 0,C 180,E1 -9795.123,E2 -9795.123} C_VEL
LIN {X 0,Y 427.009,Z 425.373,A -85,B 0,C 180,E1 -9796.093,E2 -9796.093} C_VEL
LIN {X 0,Y 426.323,Z 435.549,A -85,B 0,C 180,E1 -9797.141,E2 -9797.141} C_VEL
LIN {X 0,Y 425.75,Z 444.892,A -85,B 0,C 180,E1 -9798.334,E2 -9798.334} C_VEL
LIN {X 0,Y 425.091,Z 453.939,A -85,B 0,C 180,E1 -9799.763,E2 -9799.763} C_VEL
LIN {X 0,Y 424.693,Z 461.23,A -85,B 0,C 180,E1 -9801.195,E2 -9801.195} C_VEL
LIN {X 0,Y 424.416,Z 466.154,A -85,B 0,C 180,E1 -9802.388,E2 -9802.388} C_VEL
LIN {X 0,Y 424.241,Z 470.588,A -85,B 0,C 180,E1 -9803.702,E2 -9803.702} C_VEL
LIN {X 0,Y 424.199,Z 474.599,A -85,B 0,C 180,E1 -9805.248,E2 -9805.248} C_VEL
LIN {X 0,Y 424.098,Z 476.487,A -85,B 0,C 180,E1 -9806.199,E2 -9806.199} C_VEL
LIN {X 0,Y 424.131,Z 477.913,A -85,B 0,C 180,E1 -9807.151,E2 -9807.151} C_VEL
LIN {X 0,Y 424.129,Z 478.924,A -85,B 0,C 180,E1 -9808.101,E2 -9808.101} C_VEL
LIN {X 0,Y 424.085,Z 479.773,A -85,B 0,C 180,E1 -9810,E2 -9810} C_VEL
LIN {X 0,Y 424.088,Z 479.572,A -85,B 0,C 180,E1 -9810.95,E2 -9810.95} C_VEL
LIN {X 0,Y 424.129,Z 478.969,A -85,B 0,C 180,E1 -9811.899,E2 -9811.899} C_VEL
LIN {X 0,Y 424.131,Z 477.975,A -85,B 0,C 180,E1 -9812.85,E2 -9812.85} C_VEL
LIN {X 0,Y 424.098,Z 476.582,A -85,B 0,C 180,E1 -9813.801,E2 -9813.801} C_VEL
LIN {X 0,Y 424.206,Z 473.647,A -85,B 0,C 180,E1 -9815.228,E2 -9815.228} C_VEL
LIN {X 0,Y 424.3,Z 469.674,A -85,B 0,C 180,E1 -9816.658,E2 -9816.658} C_VEL
LIN {X 0,Y 424.582,Z 463.571,A -85,B 0,C 180,E1 -9818.328,E2 -9818.328} C_VEL
LIN {X 0,Y 424.944,Z 456.894,A -85,B 0,C 180,E1 -9819.76,E2 -9819.76} C_VEL
LIN {X 0,Y 425.475,Z 448.611,A -85,B 0,C 180,E1 -9821.191,E2 -9821.191} C_VEL
LIN {X 0,Y 426.166,Z 440.146,A -85,B 0,C 180,E1 -9822.38,E2 -9822.38} C_VEL
LIN {X 0,Y 426.866,Z 429.92,A -85,B 0,C 180,E1 -9823.546,E2 -9823.546} C_VEL
LIN {X 0,Y 427.477,Z 419.361,A -85,B 0,C 180,E1 -9824.52,E2 -9824.52} C_VEL
LIN {X 0,Y 428.192,Z 408.059,A -85,B 0,C 180,E1 -9825.347,E2 -9825.347} C_VEL
LIN {X 0,Y 428.85,Z 396.564,A -85,B 0,C 180,E1 -9825.993,E2 -9825.993} C_VEL
LIN {X 0,Y 429.378,Z 383.406,A -85,B 0,C 180,E1 -9826.523,E2 -9826.523} C_VEL
LIN {X 0,Y 429.8,Z 370.771,A -85,B 0,C 180,E1 -9826.842,E2 -9826.842} C_VEL
LIN {X 0,Y 430.53,Z 290.521,A -85,B 0,C 180,E1 -9828.221,E2 -9828.221} C_VEL
LIN {X 0,Y 426.611,Z 266.884,A -85,B 0,C 180,E1 -9828.827,E2 -9828.827} C_VEL
LIN {X 0,Y 427.672,Z 249.398,A -85,B 0,C 180,E1 -9832.208,E2 -9832.208} C_VEL
LIN {X 0,Y 428.025,Z 240.415,A -85,B 0,C 180,E1 -9833.978,E2 -9833.978} C_VEL
LIN {X 0,Y 425.815,Z 228.802,A -85,B 0,C 180,E1 -9836.464,E2 -9836.464} C_VEL
LIN {X 0,Y 425.337,Z 226.505,A -85,B 0,C 180,E1 -9836.997,E2 -9836.997} C_VEL
LIN {X 0,Y 425.292,Z 226.511,A -85,B 0,C 180,E1 -9839.719,E2 -9839.719} C_VEL
LIN {X 0,Y 425.283,Z 226.513,A -85,B 0,C 180,E1 -9843.048,E2 -9843.048} C_VEL
LIN {X 0,Y 425.282,Z 226.509,A -85,B 0,C 180,E1 -9845.928,E2 -9845.928} C_VEL
LIN {X 0,Y 425.288,Z 226.51,A -85,B 0,C 180,E1 -9849.041,E2 -9849.041} C_VEL
LIN {X 0,Y 425.291,Z 226.506,A -85,B 0,C 180,E1 -9851.958,E2 -9851.958} C_VEL
LIN {X 0,Y 425.286,Z 226.51,A -85,B 0,C 180,E1 -9855.283,E2 -9855.283} C_VEL
LIN {X 0,Y 425.274,Z 226.506,A -85,B 0,C 180,E1 -9858.621,E2 -9858.621} C_VEL
LIN {X 0,Y 425.302,Z 226.507,A -85,B 0,C 180,E1 -9861.102,E2 -9861.102} C_VEL
LIN {X 0,Y 425.3,Z 226.505,A -85,B 0,C 180,E1 -9864.664,E2 -9864.664} C_VEL
LIN {X 0,Y 425.264,Z 226.506,A -85,B 0,C 180,E1 -9868.073,E2 -9868.073} C_VEL
LIN {X 0,Y 425.331,Z 226.502,A -85,B 0,C 180,E1 -9871.368,E2 -9871.368} C_VEL
LIN {X 0,Y 425.295,Z 226.506,A -85,B 0,C 180,E1 -9874.555,E2 -9874.555} C_VEL
LIN {X 0,Y 425.287,Z 226.506,A -85,B 0,C 180,E1 -9877.661,E2 -9877.661} C_VEL
LIN {X 0,Y 425.361,Z 226.5,A -85,B 0,C 180,E1 -9880.704,E2 -9880.704} C_VEL
LIN {X 0,Y 425.388,Z 226.494,A -85,B 0,C 180,E1 -9883.688,E2 -9883.688} C_VEL
LIN {X 0,Y 425.411,Z 226.491,A -85,B 0,C 180,E1 -9887.598,E2 -9887.598} C_VEL
LIN {X 0,Y 425.442,Z 226.487,A -85,B 0,C 180,E1 -9891.45,E2 -9891.45} C_VEL
LIN {X 0,Y 425.549,Z 226.473,A -85,B 0,C 180,E1 -9894.313,E2 -9894.313} C_VEL
LIN {X 0,Y 425.575,Z 226.471,A -85,B 0,C 180,E1 -9898.107,E2 -9898.107} C_VEL
LIN {X 0,Y 425.701,Z 226.449,A -85,B 0,C 180,E1 -9900,E2 -9900} C_VEL
LIN {X 0,Y 425.554,Z 226.475,A -85,B 0,C 180,E1 -9902.84,E2 -9902.84} C_VEL
LIN {X 0,Y 425.527,Z 226.482,A -85,B 0,C 180,E1 -9906.639,E2 -9906.639} C_VEL
LIN {X 0,Y 425.4,Z 226.493,A -85,B 0,C 180,E1 -9909.509,E2 -9909.509} C_VEL
LIN {X 0,Y 425.393,Z 226.498,A -85,B 0,C 180,E1 -9912.904,E2 -9912.904} C_VEL
LIN {X 0,Y 425.361,Z 226.502,A -85,B 0,C 180,E1 -9916.605,E2 -9916.605} C_VEL
LIN {X 0,Y 425.328,Z 226.502,A -85,B 0,C 180,E1 -9919.636,E2 -9919.636} C_VEL
LIN {X 0,Y 425.287,Z 226.51,A -85,B 0,C 180,E1 -9922.339,E2 -9922.339} C_VEL
LIN {X 0,Y 425.32,Z 226.509,A -85,B 0,C 180,E1 -9924.658,E2 -9924.658} C_VEL
LIN {X 0,Y 425.299,Z 226.506,A -85,B 0,C 180,E1 -9927.561,E2 -9927.561} C_VEL
LIN {X 0,Y 425.287,Z 226.51,A -85,B 0,C 180,E1 -9930.816,E2 -9930.816} C_VEL
LIN {X 0,Y 425.309,Z 226.511,A -85,B 0,C 180,E1 -9934.288,E2 -9934.288} C_VEL
LIN {X 0,Y 425.272,Z 226.512,A -85,B 0,C 180,E1 -9937.695,E2 -9937.695} C_VEL
LIN {X 0,Y 425.244,Z 226.516,A -85,B 0,C 180,E1 -9940.515,E2 -9940.515} C_VEL
LIN {X 0,Y 425.308,Z 226.529,A -85,B 0,C 180,E1 -9942.156,E2 -9942.156} C_VEL
LIN {X 0,Y 427.203,Z 236.222,A -85,B 0,C 180,E1 -9944.34,E2 -9944.34} C_VEL
LIN {X 0,Y 426.932,Z 245.217,A -85,B 0,C 180,E1 -9946.225,E2 -9946.225} C_VEL
LIN {X 0,Y 430.879,Z 264.485,A -85,B 0,C 180,E1 -9946.772,E2 -9946.772} C_VEL
LIN {X 0,Y 429.801,Z 352.497,A -85,B 0,C 180,E1 -9948.291,E2 -9948.291} C_VEL
LIN {X 0,Y 429.413,Z 365.763,A -85,B 0,C 180,E1 -9948.704,E2 -9948.704} C_VEL
LIN {X 0,Y 428.926,Z 378.227,A -85,B 0,C 180,E1 -9949.282,E2 -9949.282} C_VEL
LIN {X 0,Y 428.308,Z 390.501,A -85,B 0,C 180,E1 -9950.06,E2 -9950.06} C_VEL
LIN {X 0,Y 427.56,Z 402.604,A -85,B 0,C 180,E1 -9951.064,E2 -9951.064} C_VEL
LIN {X 0,Y 426.913,Z 412.24,A -85,B 0,C 180,E1 -9952.065,E2 -9952.065} C_VEL
LIN {X 0,Y 426.229,Z 421.829,A -85,B 0,C 180,E1 -9953.293,E2 -9953.293} C_VEL
LIN {X 0,Y 425.599,Z 430.611,A -85,B 0,C 180,E1 -9954.693,E2 -9954.693} C_VEL
LIN {X 0,Y 425.087,Z 437.665,A -85,B 0,C 180,E1 -9956.083,E2 -9956.083} C_VEL
LIN {X 0,Y 424.711,Z 443.66,A -85,B 0,C 180,E1 -9957.558,E2 -9957.558} C_VEL
LIN {X 0,Y 424.445,Z 448.551,A -85,B 0,C 180,E1 -9959.116,E2 -9959.116} C_VEL
LIN {X 0,Y 424.25,Z 452.298,A -85,B 0,C 180,E1 -9960.746,E2 -9960.746} C_VEL
LIN {X 0,Y 424.004,Z 454.754,A -85,B 0,C 180,E1 -9962.347,E2 -9962.347} C_VEL
LIN {X 0,Y 423.944,Z 455.844,A -85,B 0,C 180,E1 -9963.534,E2 -9963.534} C_VEL
LIN {X 0,Y 423.922,Z 456.23,A -85,B 0,C 180,E1 -9964.466,E2 -9964.466} C_VEL
LIN {X 0,Y 423.904,Z 456.176,A -85,B 0,C 180,E1 -9965.764,E2 -9965.764} C_VEL
LIN {X 0,Y 423.983,Z 454.794,A -85,B 0,C 180,E1 -9967.589,E2 -9967.589} C_VEL
LIN {X 0,Y 424.105,Z 453.374,A -85,B 0,C 180,E1 -9968.619,E2 -9968.619} C_VEL
LIN {X 0,Y 424.334,Z 450.333,A -85,B 0,C 180,E1 -9970.152,E2 -9970.152} C_VEL
LIN {X 0,Y 424.529,Z 446.172,A -85,B 0,C 180,E1 -9971.667,E2 -9971.667} C_VEL
LIN {X 0,Y 424.802,Z 440.545,A -85,B 0,C 180,E1 -9973.22,E2 -9973.22} C_VEL
LIN {X 0,Y 425.25,Z 433.882,A -85,B 0,C 180,E1 -9974.667,E2 -9974.667} C_VEL
LIN {X 0,Y 425.826,Z 425.336,A -85,B 0,C 180,E1 -9976.154,E2 -9976.154} C_VEL
LIN {X 0,Y 426.159,Z 420.408,A -85,B 0,C 180,E1 -9976.873,E2 -9976.873} C_VEL
LIN {X 0,Y 425.755,Z 416.294,A -85,B 0,C 180,E1 -9977.436,E2 -9977.436} C_VEL
LIN {X 0,Y 422.344,Z 406.481,A -85,B 0,C 180,E1 -9978.686,E2 -9978.686} C_VEL
LIN {X 0,Y 420.895,Z 400.359,A -85,B 0,C 180,E1 -9979.338,E2 -9979.338} C_VEL
LIN {X 0,Y 420.832,Z 397.065,A -85,B 0,C 180,E1 -9979.634,E2 -9979.634} C_VEL
LIN {X 0,Y 421.541,Z 385.176,A -85,B 0,C 180,E1 -9980.524,E2 -9980.524} C_VEL
LIN {X 0,Y 422.066,Z 373.286,A -85,B 0,C 180,E1 -9981.2,E2 -9981.2} C_VEL
LIN {X 0,Y 422.49,Z 360.437,A -85,B 0,C 180,E1 -9981.721,E2 -9981.721} C_VEL
LIN {X 0,Y 422.825,Z 347.091,A -85,B 0,C 180,E1 -9982.058,E2 -9982.058} C_VEL
LIN {X 0,Y 423.791,Z 265.397,A -85,B 0,C 180,E1 -9983.468,E2 -9983.468} C_VEL
LIN {X 0,Y 419.903,Z 245.437,A -85,B 0,C 180,E1 -9984.025,E2 -9984.025} C_VEL
LIN {X 0,Y 420.177,Z 238.072,A -85,B 0,C 180,E1 -9985.683,E2 -9985.683} C_VEL
LIN {X 0,Y 418.526,Z 227.353,A -85,B 0,C 180,E1 -9988.256,E2 -9988.256} C_VEL
LIN {X 0,Y 418.545,Z 227.347,A -85,B 0,C 180,E1 -9990,E2 -9990} C_VEL
LIN {X 0,Y 418.476,Z 227.358,A -85,B 0,C 180,E1 -9992.888,E2 -9992.888} C_VEL
LIN {X 0,Y 418.488,Z 227.359,A -85,B 0,C 180,E1 -9995.783,E2 -9995.783} C_VEL
LIN {X 0,Y 418.38,Z 227.366,A -85,B 0,C 180,E1 -9998.695,E2 -9998.695} C_VEL
LIN {X 0,Y 418.317,Z 227.38,A -85,B 0,C 180,E1 -10001.631,E2 -10001.631} C_VEL
LIN {X 0,Y 418.3,Z 227.377,A -85,B 0,C 180,E1 -10004.597,E2 -10004.597} C_VEL
LIN {X 0,Y 418.286,Z 227.383,A -85,B 0,C 180,E1 -10007.604,E2 -10007.604} C_VEL
LIN {X 0,Y 418.252,Z 227.383,A -85,B 0,C 180,E1 -10010.663,E2 -10010.663} C_VEL
LIN {X 0,Y 418.286,Z 227.384,A -85,B 0,C 180,E1 -10013.781,E2 -10013.781} C_VEL
LIN {X 0,Y 418.228,Z 227.386,A -85,B 0,C 180,E1 -10017.048,E2 -10017.048} C_VEL
LIN {X 0,Y 418.243,Z 227.386,A -85,B 0,C 180,E1 -10020.272,E2 -10020.272} C_VEL
LIN {X 0,Y 418.249,Z 227.389,A -85,B 0,C 180,E1 -10023.677,E2 -10023.677} C_VEL
LIN {X 0,Y 418.238,Z 227.386,A -85,B 0,C 180,E1 -10027.224,E2 -10027.224} C_VEL
LIN {X 0,Y 418.242,Z 227.39,A -85,B 0,C 180,E1 -10029.683,E2 -10029.683} C_VEL
LIN {X 0,Y 418.223,Z 227.389,A -85,B 0,C 180,E1 -10032.32,E2 -10032.32} C_VEL
LIN {X 0,Y 418.235,Z 227.386,A -85,B 0,C 180,E1 -10035.108,E2 -10035.108} C_VEL
LIN {X 0,Y 418.239,Z 227.39,A -85,B 0,C 180,E1 -10037.766,E2 -10037.766} C_VEL
LIN {X 0,Y 418.248,Z 227.386,A -85,B 0,C 180,E1 -10040.62,E2 -10040.62} C_VEL
LIN {X 0,Y 418.243,Z 227.388,A -85,B 0,C 180,E1 -10043.975,E2 -10043.975} C_VEL
LIN {X 0,Y 418.256,Z 227.384,A -85,B 0,C 180,E1 -10047.156,E2 -10047.156} C_VEL
LIN {X 0,Y 418.267,Z 227.383,A -85,B 0,C 180,E1 -10050.895,E2 -10050.895} C_VEL
LIN {X 0,Y 418.269,Z 227.384,A -85,B 0,C 180,E1 -10054.096,E2 -10054.096} C_VEL
LIN {X 0,Y 418.236,Z 227.387,A -85,B 0,C 180,E1 -10057.264,E2 -10057.264} C_VEL
LIN {X 0,Y 418.281,Z 227.383,A -85,B 0,C 180,E1 -10060.364,E2 -10060.364} C_VEL
LIN {X 0,Y 418.315,Z 227.377,A -85,B 0,C 180,E1 -10063.404,E2 -10063.404} C_VEL
LIN {X 0,Y 418.344,Z 227.373,A -85,B 0,C 180,E1 -10066.999,E2 -10066.999} C_VEL
LIN {X 0,Y 418.339,Z 227.376,A -85,B 0,C 180,E1 -10070.328,E2 -10070.328} C_VEL
LIN {X 0,Y 418.492,Z 227.355,A -85,B 0,C 180,E1 -10073.249,E2 -10073.249} C_VEL
LIN {X 0,Y 418.338,Z 227.374,A -85,B 0,C 180,E1 -10075.181,E2 -10075.181} C_VEL
LIN {X 0,Y 418.542,Z 227.35,A -85,B 0,C 180,E1 -10078.075,E2 -10078.075} C_VEL
LIN {X 0,Y 418.668,Z 227.334,A -85,B 0,C 180,E1 -10080,E2 -10080} C_VEL
LIN {X 0,Y 418.508,Z 227.353,A -85,B 0,C 180,E1 -10082.888,E2 -10082.888} C_VEL
LIN {X 0,Y 418.491,Z 227.356,A -85,B 0,C 180,E1 -10086.751,E2 -10086.751} C_VEL
LIN {X 0,Y 418.338,Z 227.375,A -85,B 0,C 180,E1 -10089.671,E2 -10089.671} C_VEL
LIN {X 0,Y 418.343,Z 227.373,A -85,B 0,C 180,E1 -10093.001,E2 -10093.001} C_VEL
LIN {X 0,Y 418.31,Z 227.379,A -85,B 0,C 180,E1 -10096.736,E2 -10096.736} C_VEL
LIN {X 0,Y 418.268,Z 227.383,A -85,B 0,C 180,E1 -10099.791,E2 -10099.791} C_VEL
LIN {X 0,Y 418.236,Z 227.388,A -85,B 0,C 180,E1 -10102.736,E2 -10102.736} C_VEL
LIN {X 0,Y 418.268,Z 227.383,A -85,B 0,C 180,E1 -10105.904,E2 -10105.904} C_VEL
LIN {X 0,Y 418.262,Z 227.382,A -85,B 0,C 180,E1 -10109.162,E2 -10109.162} C_VEL
LIN {X 0,Y 418.255,Z 227.385,A -85,B 0,C 180,E1 -10112.844,E2 -10112.844} C_VEL
LIN {X 0,Y 418.244,Z 227.387,A -85,B 0,C 180,E1 -10116.238,E2 -10116.238} C_VEL
LIN {X 0,Y 418.247,Z 227.384,A -85,B 0,C 180,E1 -10119.683,E2 -10119.683} C_VEL
LIN {X 0,Y 418.228,Z 227.39,A -85,B 0,C 180,E1 -10122.322,E2 -10122.322} C_VEL
LIN {X 0,Y 418.234,Z 227.386,A -85,B 0,C 180,E1 -10125.109,E2 -10125.109} C_VEL
LIN {X 0,Y 418.239,Z 227.385,A -85,B 0,C 180,E1 -10127.767,E2 -10127.767} C_VEL
LIN {X 0,Y 418.254,Z 227.387,A -85,B 0,C 180,E1 -10130.619,E2 -10130.619} C_VEL
LIN {X 0,Y 418.241,Z 227.385,A -85,B 0,C 180,E1 -10133.976,E2 -10133.976} C_VEL
LIN {X 0,Y 418.258,Z 227.387,A -85,B 0,C 180,E1 -10137.156,E2 -10137.156} C_VEL
LIN {X 0,Y 418.269,Z 227.386,A -85,B 0,C 180,E1 -10140.896,E2 -10140.896} C_VEL
LIN {X 0,Y 418.346,Z 227.557,A -85,B 0,C 180,E1 -10142.783,E2 -10142.783} C_VEL
LIN {X 0,Y 421.067,Z 241.519,A -85,B 0,C 180,E1 -10145.863,E2 -10145.863} C_VEL
LIN {X 0,Y 420.912,Z 247.227,A -85,B 0,C 180,E1 -10147.028,E2 -10147.028} C_VEL
LIN {X 0,Y 419.891,Z 263.166,A -85,B 0,C 180,E1 -10150.214,E2 -10150.214} C_VEL
LIN {X 0,Y 419.596,Z 267.218,A -85,B 0,C 180,E1 -10151.015,E2 -10151.015} C_VEL
LIN {X 0,Y 423.604,Z 293.033,A -85,B 0,C 180,E1 -10151.656,E2 -10151.656} C_VEL
LIN {X 0,Y 422.589,Z 375.955,A -85,B 0,C 180,E1 -10153.111,E2 -10153.111} C_VEL
LIN {X 0,Y 422.089,Z 389.748,A -85,B 0,C 180,E1 -10153.557,E2 -10153.557} C_VEL
LIN {X 0,Y 421.495,Z 402.149,A -85,B 0,C 180,E1 -10154.155,E2 -10154.155} C_VEL
LIN {X 0,Y 420.824,Z 413.238,A -85,B 0,C 180,E1 -10154.874,E2 -10154.874} C_VEL
LIN {X 0,Y 420.128,Z 424.348,A -85,B 0,C 180,E1 -10155.795,E2 -10155.795} C_VEL
LIN {X 0,Y 419.381,Z 435.244,A -85,B 0,C 180,E1 -10156.925,E2 -10156.925} C_VEL
LIN {X 0,Y 418.759,Z 444.618,A -85,B 0,C 180,E1 -10158.136,E2 -10158.136} C_VEL
LIN {X 0,Y 418.059,Z 453.682,A -85,B 0,C 180,E1 -10159.589,E2 -10159.589} C_VEL
LIN {X 0,Y 417.649,Z 460.987,A -85,B 0,C 180,E1 -10161.045,E2 -10161.045} C_VEL
LIN {X 0,Y 417.356,Z 465.922,A -85,B 0,C 180,E1 -10162.258,E2 -10162.258} C_VEL
LIN {X 0,Y 417.166,Z 470.7,A -85,B 0,C 180,E1 -10163.709,E2 -10163.709} C_VEL
LIN {X 0,Y 417.106,Z 474.382,A -85,B 0,C 180,E1 -10165.167,E2 -10165.167} C_VEL
LIN {X 0,Y 417.013,Z 476.274,A -85,B 0,C 180,E1 -10166.135,E2 -10166.135} C_VEL
LIN {X 0,Y 417.028,Z 477.706,A -85,B 0,C 180,E1 -10167.102,E2 -10167.102} C_VEL
LIN {X 0,Y 417.056,Z 478.721,A -85,B 0,C 180,E1 -10168.069,E2 -10168.069} C_VEL
LIN {X 0,Y 417.005,Z 479.576,A -85,B 0,C 180,E1 -10170,E2 -10170} C_VEL
LIN {X 0,Y 417.011,Z 479.38,A -85,B 0,C 180,E1 -10170.966,E2 -10170.966} C_VEL
LIN {X 0,Y 417.056,Z 478.779,A -85,B 0,C 180,E1 -10171.932,E2 -10171.932} C_VEL
LIN {X 0,Y 417.027,Z 477.786,A -85,B 0,C 180,E1 -10172.898,E2 -10172.898} C_VEL
LIN {X 0,Y 417.013,Z 476.396,A -85,B 0,C 180,E1 -10173.866,E2 -10173.866} C_VEL
LIN {X 0,Y 417.121,Z 473.465,A -85,B 0,C 180,E1 -10175.317,E2 -10175.317} C_VEL
LIN {X 0,Y 417.233,Z 469.499,A -85,B 0,C 180,E1 -10176.772,E2 -10176.772} C_VEL
LIN {X 0,Y 417.523,Z 463.409,A -85,B 0,C 180,E1 -10178.47,E2 -10178.47} C_VEL
LIN {X 0,Y 417.925,Z 456.743,A -85,B 0,C 180,E1 -10179.926,E2 -10179.926} C_VEL
LIN {X 0,Y 418.498,Z 448.475,A -85,B 0,C 180,E1 -10181.38,E2 -10181.38} C_VEL
LIN {X 0,Y 419.203,Z 440.023,A -85,B 0,C 180,E1 -10182.589,E2 -10182.589} C_VEL
LIN {X 0,Y 419.889,Z 429.619,A -85,B 0,C 180,E1 -10183.796,E2 -10183.796} C_VEL
LIN {X 0,Y 420.69,Z 417.851,A -85,B 0,C 180,E1 -10184.883,E2 -10184.883} C_VEL
LIN {X 0,Y 421.458,Z 406.146,A -85,B 0,C 180,E1 -10185.722,E2 -10185.722} C_VEL
LIN {X 0,Y 422.184,Z 393.999,A -85,B 0,C 180,E1 -10186.377,E2 -10186.377} C_VEL
